# B&R Automation Studio project DivDiag
Automation Studio 4.9.2.46; technology packages: mapp 5.14.0, mappCockpit 5.14.0, mappMotion 5.14.0, mappView 5.14.0

## Configuration APC_XRAY

CPU PC_any, AutomationRuntime C4.72, Build 4.1.2, Safety 0.0, Vc V4.72.0

### Task classes (Cpu.sw)
```
Cyclic#1 (cycle 1600 us, tolerance 0 us):
  MainTest <- Source.MainTest.prg
  Maint <- Source.Diagnostic.Maint.prg
Cyclic#8 (cycle 9600 us):
  Vis <- Source.Vis.prg
DataObjects: McAcpSys
Binaries: mCoWebSc, FWRules, TCData, udbdef, mvLoader, McAcpSim, arsvcreg, McAcpDrv, arflatprv, arcoal, arconfig, Role, User, Cfg_Sec, asfw, iomap, Cfg_Sh, ashwd, ashwac, Cfg_PpList, sysconf, Cfg_Trak, McProfGen, TCLang, Cfg_Aut, Cfg_PVirt, Cfg_Ax, asnxdb1, Settings, CfgRec, Cfg_App2, Cfg_Comp, Cfg_Auto, Cfg_App1, Cfg_Set, TC, asnxdb2, AlarmCfg, AlarmHist, SSLCfg, Cfg_App6, Cfg_App5, Cfg_App4, Cfg_App3, AuditCfg, Cfg_Coupl, vccdt, vccline, vcfile, arial, vccbmp, vccstr, vcctrend, vcbclass, vcgclass, vcdsint, vcnet, vcshared, vcmgr, arialbd, vcxml, vccnum, vccbtn, vccovl, vccalarm, vccurl, vccslider, vccbar, vcctext, Visu01, Visu03, vcpdsw, vcfntttf, vcalarm, Visu02, vcrt, vcchtml, vcdsloc, vcchspot, vctcal, vcpdvnc, vcpfar00, vcpfmtcx, vcptelo, vcpdihd, vcpdi855, vcpfapc, vcpfppc7, vcpdi815, vcpk, Config_1, Config_4, Config_3, Config_2, CfgAlrm
Libraries: standard, AsBrStr, McAcpPar, McBase, sys_lib, runtime, arssl, fileio, mcacptrak, astime, asieccon, powerlnk, mcaxis, dataobj, aruser, mpaudit, vcresman, AsIODiag
```

### Hardware
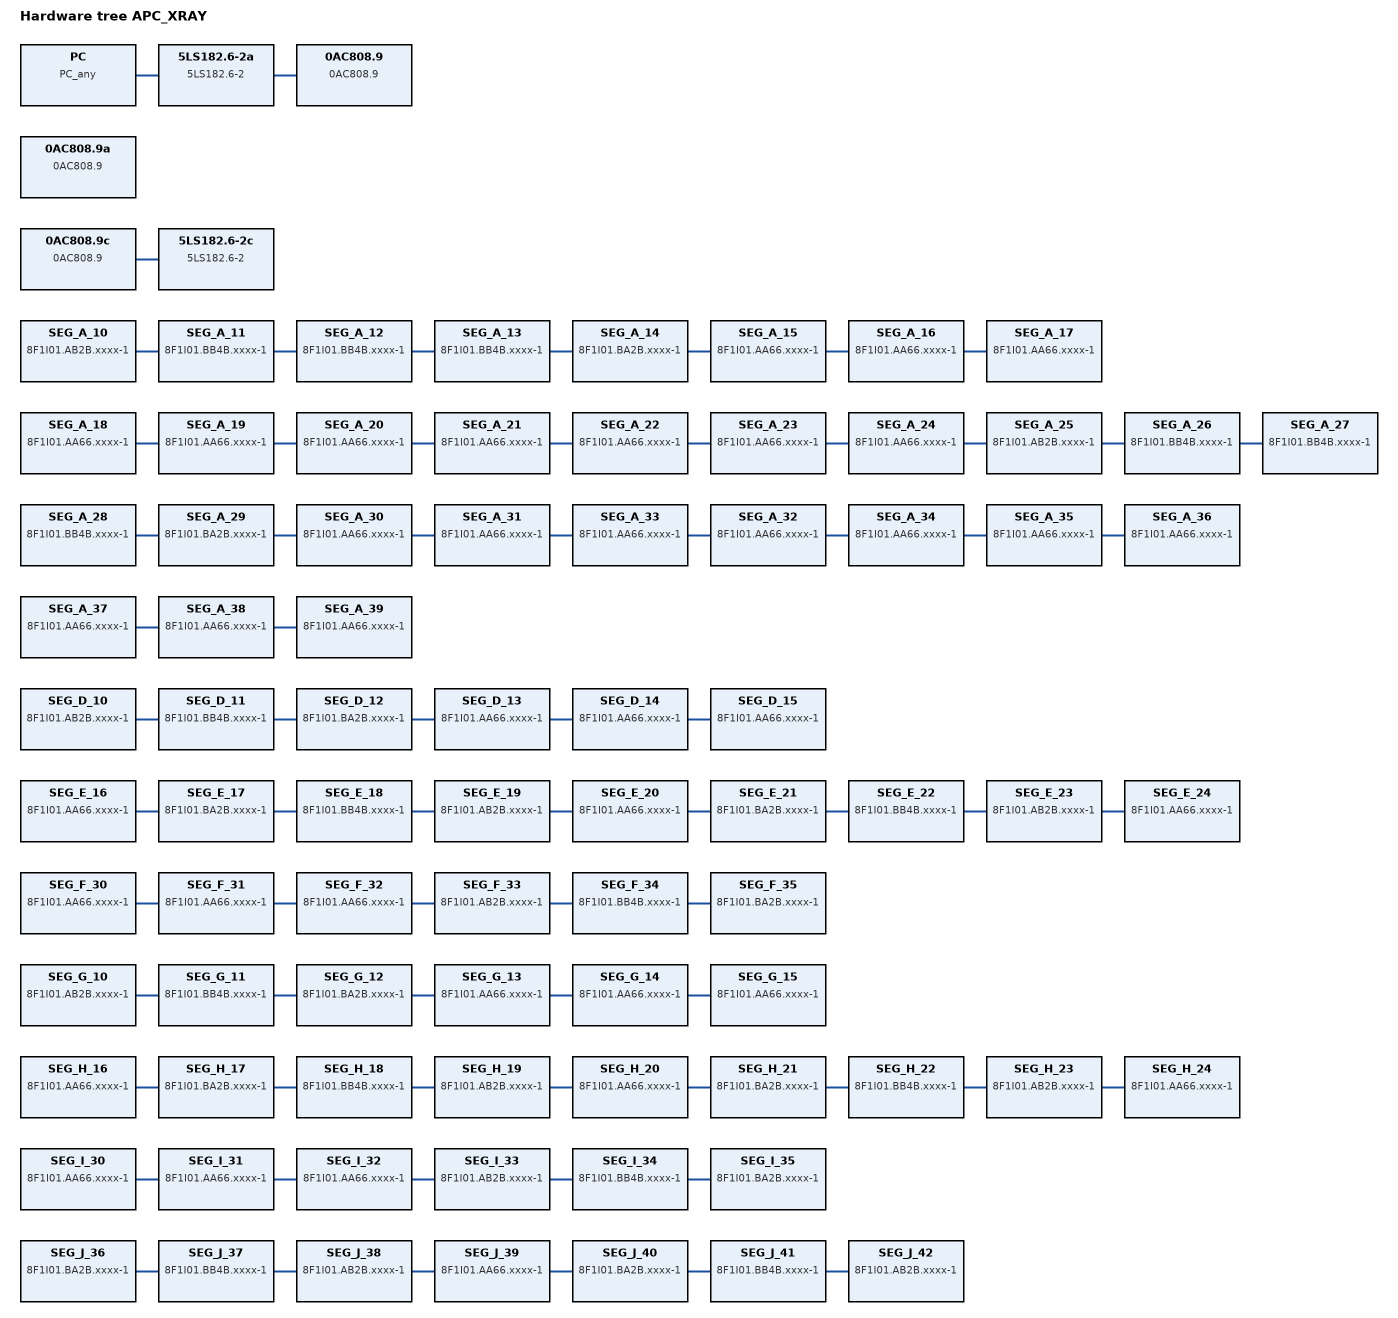
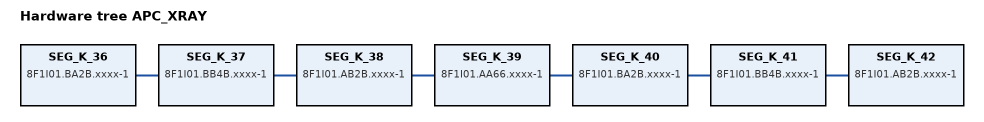
```
0AC808.9 : 0AC808.9 v1.0.0.0  [ETH1 -> 5LS182.6-2a.IF1 [Cable Type=PowerlinkCable, Length=10, Version=1.0.0.3]; ETH2 -> SEG_A_12.PLK3 [Cable Type=PowerlinkCable, Length=10, Version=1.0.0.3]; ETH3 -> SEG_A_22.PLK3 [Cable Type=PowerlinkCable, Length=10, Version=1.0.0.3]; ETH4 -> SEG_A_32.PLK3 [Cable Type=PowerlinkCable, Length=10, Version=1.0.0.3]]
0AC808.9a : 0AC808.9 v1.0.0.0  [ETH1 -> 5LS182.6-2c.IF1 [Cable Type=PowerlinkCable, Length=10, Version=1.0.0.3]; ETH2 -> SEG_G_10.PLK3 [Cable Type=PowerlinkCable, Length=10, Version=1.0.0.3]; ETH3 -> SEG_H_20.PLK3 [Cable Type=PowerlinkCable, Length=10, Version=1.0.0.3]; ETH4 -> SEG_I_35.PLK3 [Cable Type=PowerlinkCable, Length=10, Version=1.0.0.3]; ETH6 -> SEG_K_39.PLK3 [Cable Type=PowerlinkCable, Length=10, Version=1.0.0.3]]
0AC808.9c : 0AC808.9 v1.0.0.0  [ETH1 -> 5LS182.6-2c.PLK2 [Cable Type=PowerlinkCable, Length=10, Version=1.0.0.3]; ETH2 -> SEG_D_10.PLK3 [Cable Type=PowerlinkCable, Length=10, Version=1.0.0.3]; ETH3 -> SEG_E_20.PLK3 [Cable Type=PowerlinkCable, Length=10, Version=1.0.0.3]; ETH4 -> SEG_F_35.PLK3 [Cable Type=PowerlinkCable, Length=10, Version=1.0.0.3]; ETH6 -> SEG_J_39.PLK3 [Cable Type=PowerlinkCable, Length=10, Version=1.0.0.3]]
5LS182.6-2a : 5LS182.6-2 v1.7.1.0  [SL -> PC.SL1]
  Connector IF1:
    MtuSize = 1500
    DNAConfiguration = manual
    CycleTime = 1600
    EplNatSubnet = 192.168.102.0
  Supervision = off
5LS182.6-2c : 5LS182.6-2 v1.7.1.0  [PLK2 -> 0AC808.9c.ETH1 [Cable Type=PowerlinkCable, Length=10, Version=1.0.0.3]; SL -> PC.SL2]
  Connector IF1:
    DNAConfiguration = manual
    CycleTime = 1600
    NodeDefinition = Software
    EplNatSubnet = 192.168.104.0
PC : PC_any v1.1.1.0 (OrderNumber=PC)
  Connector IF1:
    ActivateDevice = 1
    ActivateIna = 1
    DeviceParam = /IR=4 /IO=0x3F8 /CLK=1843200 /IF=1
  Connector IF3:
    InaPort = 11159
  ConfigurationID = Starwheel_XRAY
  ConfigVersion = 1.0.2
  UserPartitionSize = 100
  UserRamSize = 250000
  RemMemSize = 250000
  PermanentPvSize = 10000
  RemanentGlobalPvSize = 10000
  VolatileGlobalPvSize = 100000
  SystemTick = 1600
  TaskClassIdleTime = 1600
  Cyclic1Duration = 1600
  Cyclic1Tolerance = 0
  Cyclic1Stack = 256000
  Cyclic2Duration = 19200
  Cyclic2Tolerance = 19200
  Cyclic3Duration = 49600
  Cyclic3Tolerance = 49600
  Cyclic4Duration = 99200
  Cyclic4Tolerance = 99200
  Cyclic6Duration = 499200
  Cyclic6Tolerance = 499200
  Cyclic8Duration = 9600
  FileDevice1
  FileDeviceName1 = SvgData
  FileDevicePath1 = ../../../../Logical/Scene/Generated
  FtpUser1
  FtpUsername1 = BnR
  FtpUserPassword1 = OwgnRUL028A/e+iGXLfM2NhZbf3ZfVOTPAeyn0eidZE=  // password
  FtpUserSalt1 = LWczKOmt
  FTPAccessRight1 = 0
  ActivateOpcUa = 1
  OpcUaInformationModels_PV_Version = 1
SEG_A_10 : 8F1I01.AB2B.xxxx-1 v1.0.0.2  [PLK1 -> SEG_A_39.PLK2 (NodeNumber=10) [Cable Type=PowerlinkCable, Length=10, Version=1.0.0.3]; PLK2 -> SEG_A_11.PLK1 (NodeNumber=10) [Cable Type=PowerlinkCable, Length=10, Version=1.0.0.3]]
  EnableDNA = on
  EPL_DNA_Head = 0
  EPL_DNA_Predecessor = 11
  EPL_DNA_HubPort = 1
  EPL_DNA_InPort = 2
  DriveConfiguration:
    McTypeID = LLMConfig
  DriveConfiguration/Segment:
    Shape = STRAIGHT105_TO_CIRCULAR
    SegmentReference = SEG_A_10
    StopReaction = UseAssemblySetting
    SpeedFilter = UseAssemblySetting
SEG_A_11 : 8F1I01.BB4B.xxxx-1 v1.0.0.2  [PLK1 -> SEG_A_10.PLK2 (NodeNumber=11) [Cable Type=PowerlinkCable, Length=10, Version=1.0.0.3]; PLK2 -> SEG_A_12.PLK1 (NodeNumber=11) [Cable Type=PowerlinkCable, Length=10, Version=1.0.0.3]]
  EnableDNA = on
  EPL_DNA_Head = 0
  EPL_DNA_Predecessor = 12
  EPL_DNA_HubPort = 1
  EPL_DNA_InPort = 2
  DriveConfiguration:
    McTypeID = LLMConfig
  DriveConfiguration/Segment:
    Shape = CIRCULAR
    SegmentReference = SEG_A_11
    StopReaction = UseAssemblySetting
    SpeedFilter = UseAssemblySetting
SEG_A_12 : 8F1I01.BB4B.xxxx-1 v1.0.0.2  [PLK1 -> SEG_A_11.PLK2 (NodeNumber=12) [Cable Type=PowerlinkCable, Length=10, Version=1.0.0.3]; PLK2 -> SEG_A_13.PLK1 (NodeNumber=12) [Cable Type=PowerlinkCable, Length=10, Version=1.0.0.3]; PLK3 -> 0AC808.9.ETH2 (NodeNumber=12) [Cable Type=PowerlinkCable, Length=10, Version=1.0.0.3]]
  EnableDNA = on
  EPL_DNA_Head = 0
  EPL_DNA_HubPort = 0
  EPL_DNA_InPort = 3
  DriveConfiguration:
    McTypeID = LLMConfig
  DriveConfiguration/Segment:
    Shape = CIRCULAR
    SegmentReference = SEG_A_12
    StopReaction = UseAssemblySetting
    SpeedFilter = UseAssemblySetting
SEG_A_13 : 8F1I01.BB4B.xxxx-1 v1.0.0.2  [PLK1 -> SEG_A_12.PLK2 (NodeNumber=13) [Cable Type=PowerlinkCable, Length=10, Version=1.0.0.3]; PLK2 -> SEG_A_14.PLK1 (NodeNumber=13) [Cable Type=PowerlinkCable, Length=10, Version=1.0.0.3]]
  EnableDNA = on
  EPL_DNA_Head = 0
  EPL_DNA_Predecessor = 12
  DriveConfiguration:
    McTypeID = LLMConfig
  DriveConfiguration/Segment:
    Shape = CIRCULAR
    SegmentReference = SEG_A_13
    StopReaction = UseAssemblySetting
    SpeedFilter = UseAssemblySetting
SEG_A_14 : 8F1I01.BA2B.xxxx-1 v1.0.0.2  [PLK1 -> SEG_A_13.PLK2 (NodeNumber=14) [Cable Type=PowerlinkCable, Length=10, Version=1.0.0.3]; PLK2 -> SEG_A_15.PLK1 (NodeNumber=14) [Cable Type=PowerlinkCable, Length=10, Version=1.0.0.3]]
  EnableDNA = on
  EPL_DNA_Head = 0
  EPL_DNA_Predecessor = 13
  DriveConfiguration:
    McTypeID = LLMConfig
  DriveConfiguration/Segment:
    Shape = CIRCULAR_TO_STRAIGHT105
    SegmentReference = SEG_A_14
    StopReaction = UseAssemblySetting
    SpeedFilter = UseAssemblySetting
SEG_A_15 : 8F1I01.AA66.xxxx-1 v1.0.0.2  [PLK1 -> SEG_A_14.PLK2 (NodeNumber=15) [Cable Type=PowerlinkCable, Length=10, Version=1.0.0.3]; PLK2 -> SEG_A_16.PLK1 (NodeNumber=15) [Cable Type=PowerlinkCable, Length=10, Version=1.0.0.3]]
  EnableDNA = on
  EPL_DNA_Head = 0
  EPL_DNA_Predecessor = 14
  DriveConfiguration:
    McTypeID = LLMConfig
  DriveConfiguration/Segment:
    Shape = STRAIGHT660
    SegmentReference = SEG_A_15
    StopReaction = UseAssemblySetting
    SpeedFilter = UseAssemblySetting
SEG_A_16 : 8F1I01.AA66.xxxx-1 v1.0.0.2  [PLK1 -> SEG_A_15.PLK2 (NodeNumber=16) [Cable Type=PowerlinkCable, Length=10, Version=1.0.0.3]; PLK2 -> SEG_A_17.PLK1 (NodeNumber=16) [Cable Type=PowerlinkCable, Length=10, Version=1.0.0.3]]
  EnableDNA = on
  EPL_DNA_Head = 0
  EPL_DNA_Predecessor = 15
  DriveConfiguration:
    McTypeID = LLMConfig
  DriveConfiguration/Segment:
    Shape = STRAIGHT660
    SegmentReference = SEG_A_16
    StopReaction = UseAssemblySetting
    SpeedFilter = UseAssemblySetting
SEG_A_17 : 8F1I01.AA66.xxxx-1 v1.0.0.2  [PLK1 -> SEG_A_16.PLK2 (NodeNumber=17) [Cable Type=PowerlinkCable, Length=10, Version=1.0.0.3]]
  EnableDNA = on
  EPL_DNA_Head = 0
  EPL_DNA_Predecessor = 16
  DriveConfiguration:
    McTypeID = LLMConfig
  DriveConfiguration/Segment:
    Shape = STRAIGHT660
    SegmentReference = SEG_A_17
    StopReaction = UseAssemblySetting
    SpeedFilter = UseAssemblySetting
SEG_A_18 : 8F1I01.AA66.xxxx-1 v1.0.0.2  [PLK2 -> SEG_A_19.PLK1 (NodeNumber=18) [Cable Type=PowerlinkCable, Length=10, Version=1.0.0.3]]
  EnableDNA = on
  EPL_DNA_Head = 0
  EPL_DNA_Predecessor = 19
  EPL_DNA_HubPort = 1
  EPL_DNA_InPort = 2
  DriveConfiguration:
    McTypeID = LLMConfig
  DriveConfiguration/Segment:
    Shape = STRAIGHT660
    SegmentReference = SEG_A_18
    StopReaction = UseAssemblySetting
    SpeedFilter = UseAssemblySetting
SEG_A_19 : 8F1I01.AA66.xxxx-1 v1.0.0.2  [PLK1 -> SEG_A_18.PLK2 (NodeNumber=19) [Cable Type=PowerlinkCable, Length=10, Version=1.0.0.3]; PLK2 -> SEG_A_20.PLK1 (NodeNumber=19) [Cable Type=PowerlinkCable, Length=10, Version=1.0.0.3]]
  EnableDNA = on
  EPL_DNA_Head = 0
  EPL_DNA_Predecessor = 20
  EPL_DNA_HubPort = 1
  EPL_DNA_InPort = 2
  DriveConfiguration:
    McTypeID = LLMConfig
  DriveConfiguration/Segment:
    Shape = STRAIGHT660
    SegmentReference = SEG_A_19
    StopReaction = UseAssemblySetting
    SpeedFilter = UseAssemblySetting
SEG_A_20 : 8F1I01.AA66.xxxx-1 v1.0.0.2  [PLK1 -> SEG_A_19.PLK2 (NodeNumber=20) [Cable Type=PowerlinkCable, Length=10, Version=1.0.0.3]; PLK2 -> SEG_A_21.PLK1 (NodeNumber=20) [Cable Type=PowerlinkCable, Length=10, Version=1.0.0.3]]
  EnableDNA = on
  EPL_DNA_Head = 0
  EPL_DNA_Predecessor = 21
  EPL_DNA_HubPort = 1
  EPL_DNA_InPort = 2
  DriveConfiguration:
    McTypeID = LLMConfig
  DriveConfiguration/Segment:
    Shape = STRAIGHT660
    SegmentReference = SEG_A_20
    StopReaction = UseAssemblySetting
    SpeedFilter = UseAssemblySetting
SEG_A_21 : 8F1I01.AA66.xxxx-1 v1.0.0.2  [PLK1 -> SEG_A_20.PLK2 (NodeNumber=21) [Cable Type=PowerlinkCable, Length=10, Version=1.0.0.3]; PLK2 -> SEG_A_22.PLK1 (NodeNumber=21) [Cable Type=PowerlinkCable, Length=10, Version=1.0.0.3]]
  EnableDNA = on
  EPL_DNA_Head = 0
  EPL_DNA_Predecessor = 22
  EPL_DNA_HubPort = 1
  EPL_DNA_InPort = 2
  DriveConfiguration:
    McTypeID = LLMConfig
  DriveConfiguration/Segment:
    Shape = STRAIGHT660
    SegmentReference = SEG_A_21
    StopReaction = UseAssemblySetting
    SpeedFilter = UseAssemblySetting
SEG_A_22 : 8F1I01.AA66.xxxx-1 v1.0.0.2  [PLK1 -> SEG_A_21.PLK2 (NodeNumber=22) [Cable Type=PowerlinkCable, Length=10, Version=1.0.0.3]; PLK2 -> SEG_A_23.PLK1 (NodeNumber=22) [Cable Type=PowerlinkCable, Length=10, Version=1.0.0.3]; PLK3 -> 0AC808.9.ETH3 (NodeNumber=22) [Cable Type=PowerlinkCable, Length=10, Version=1.0.0.3]]
  EnableDNA = on
  EPL_DNA_Head = 0
  EPL_DNA_HubPort = 0
  EPL_DNA_InPort = 3
  DriveConfiguration:
    McTypeID = LLMConfig
  DriveConfiguration/Segment:
    Shape = STRAIGHT660
    SegmentReference = SEG_A_22
    StopReaction = UseAssemblySetting
    SpeedFilter = UseAssemblySetting
SEG_A_23 : 8F1I01.AA66.xxxx-1 v1.0.0.2  [PLK1 -> SEG_A_22.PLK2 (NodeNumber=23) [Cable Type=PowerlinkCable, Length=10, Version=1.0.0.3]; PLK2 -> SEG_A_24.PLK1 (NodeNumber=23) [Cable Type=PowerlinkCable, Length=10, Version=1.0.0.3]]
  EnableDNA = on
  EPL_DNA_Head = 0
  EPL_DNA_Predecessor = 22
  DriveConfiguration:
    McTypeID = LLMConfig
  DriveConfiguration/Segment:
    Shape = STRAIGHT660
    SegmentReference = SEG_A_23
    StopReaction = UseAssemblySetting
    SpeedFilter = UseAssemblySetting
SEG_A_24 : 8F1I01.AA66.xxxx-1 v1.0.0.2  [PLK1 -> SEG_A_23.PLK2 (NodeNumber=24) [Cable Type=PowerlinkCable, Length=10, Version=1.0.0.3]; PLK2 -> SEG_A_25.PLK1 (NodeNumber=24) [Cable Type=PowerlinkCable, Length=10, Version=1.0.0.3]]
  EnableDNA = on
  EPL_DNA_Head = 0
  EPL_DNA_Predecessor = 23
  DriveConfiguration:
    McTypeID = LLMConfig
  DriveConfiguration/Segment:
    Shape = STRAIGHT660
    SegmentReference = SEG_A_24
    StopReaction = UseAssemblySetting
    SpeedFilter = UseAssemblySetting
SEG_A_25 : 8F1I01.AB2B.xxxx-1 v1.0.0.2  [PLK1 -> SEG_A_24.PLK2 (NodeNumber=25) [Cable Type=PowerlinkCable, Length=10, Version=1.0.0.3]; PLK2 -> SEG_A_26.PLK1 (NodeNumber=25) [Cable Type=PowerlinkCable, Length=10, Version=1.0.0.3]]
  EnableDNA = on
  EPL_DNA_Head = 0
  EPL_DNA_Predecessor = 24
  DriveConfiguration:
    McTypeID = LLMConfig
  DriveConfiguration/Segment:
    Shape = STRAIGHT105_TO_CIRCULAR
    SegmentReference = SEG_A_25
    StopReaction = UseAssemblySetting
    SpeedFilter = UseAssemblySetting
SEG_A_26 : 8F1I01.BB4B.xxxx-1 v1.0.0.2  [PLK1 -> SEG_A_25.PLK2 (NodeNumber=26) [Cable Type=PowerlinkCable, Length=10, Version=1.0.0.3]; PLK2 -> SEG_A_27.PLK1 (NodeNumber=26) [Cable Type=PowerlinkCable, Length=10, Version=1.0.0.3]]
  EnableDNA = on
  EPL_DNA_Head = 0
  EPL_DNA_Predecessor = 25
  DriveConfiguration:
    McTypeID = LLMConfig
  DriveConfiguration/Segment:
    Shape = CIRCULAR
    SegmentReference = SEG_A_26
    StopReaction = UseAssemblySetting
    SpeedFilter = UseAssemblySetting
SEG_A_27 : 8F1I01.BB4B.xxxx-1 v1.0.0.2  [PLK1 -> SEG_A_26.PLK2 (NodeNumber=27) [Cable Type=PowerlinkCable, Length=10, Version=1.0.0.3]]
  EnableDNA = on
  EPL_DNA_Head = 0
  EPL_DNA_Predecessor = 26
  DriveConfiguration:
    McTypeID = LLMConfig
  DriveConfiguration/Segment:
    Shape = CIRCULAR
    SegmentReference = SEG_A_27
    StopReaction = UseAssemblySetting
    SpeedFilter = UseAssemblySetting
SEG_A_28 : 8F1I01.BB4B.xxxx-1 v1.0.0.2  [PLK2 -> SEG_A_29.PLK1 (NodeNumber=28) [Cable Type=PowerlinkCable, Length=10, Version=1.0.0.3]]
  EnableDNA = on
  EPL_DNA_Head = 0
  EPL_DNA_Predecessor = 29
  EPL_DNA_HubPort = 1
  EPL_DNA_InPort = 2
  DriveConfiguration:
    McTypeID = LLMConfig
  DriveConfiguration/Segment:
    Shape = CIRCULAR
    SegmentReference = SEG_A_28
    StopReaction = UseAssemblySetting
    SpeedFilter = UseAssemblySetting
SEG_A_29 : 8F1I01.BA2B.xxxx-1 v1.0.0.2  [PLK1 -> SEG_A_28.PLK2 (NodeNumber=29) [Cable Type=PowerlinkCable, Length=10, Version=1.0.0.3]; PLK2 -> SEG_A_30.PLK1 (NodeNumber=29) [Cable Type=PowerlinkCable, Length=10, Version=1.0.0.3]]
  EnableDNA = on
  EPL_DNA_Head = 0
  EPL_DNA_Predecessor = 30
  EPL_DNA_HubPort = 1
  EPL_DNA_InPort = 2
  DriveConfiguration:
    McTypeID = LLMConfig
  DriveConfiguration/Segment:
    Shape = CIRCULAR_TO_STRAIGHT105
    SegmentReference = SEG_A_29
    StopReaction = UseAssemblySetting
    SpeedFilter = UseAssemblySetting
SEG_A_30 : 8F1I01.AA66.xxxx-1 v1.0.0.2  [PLK1 -> SEG_A_29.PLK2 (NodeNumber=30) [Cable Type=PowerlinkCable, Length=10, Version=1.0.0.3]; PLK2 -> SEG_A_31.PLK1 (NodeNumber=30) [Cable Type=PowerlinkCable, Length=10, Version=1.0.0.3]]
  EnableDNA = on
  EPL_DNA_Head = 0
  EPL_DNA_Predecessor = 31
  EPL_DNA_HubPort = 1
  EPL_DNA_InPort = 2
  DriveConfiguration:
    McTypeID = LLMConfig
  DriveConfiguration/Segment:
    Shape = STRAIGHT660
    SegmentReference = SEG_A_30
    StopReaction = UseAssemblySetting
    SpeedFilter = UseAssemblySetting
SEG_A_31 : 8F1I01.AA66.xxxx-1 v1.0.0.2  [PLK1 -> SEG_A_30.PLK2 (NodeNumber=31) [Cable Type=PowerlinkCable, Length=10, Version=1.0.0.3]; PLK2 -> SEG_A_33.PLK1 (NodeNumber=31) [Cable Type=PowerlinkCable, Length=10, Version=1.0.0.3]]
  EnableDNA = on
  EPL_DNA_Head = 0
  EPL_DNA_Predecessor = 32
  EPL_DNA_HubPort = 1
  EPL_DNA_InPort = 2
  DriveConfiguration:
    McTypeID = LLMConfig
  DriveConfiguration/Segment:
    Shape = STRAIGHT660
    SegmentReference = SEG_A_31
    StopReaction = UseAssemblySetting
    SpeedFilter = UseAssemblySetting
SEG_A_32 : 8F1I01.AA66.xxxx-1 v1.0.0.2  [PLK1 -> SEG_A_33.PLK2 (NodeNumber=32) [Cable Type=PowerlinkCable, Length=10, Version=1.0.0.3]; PLK2 -> SEG_A_34.PLK1 (NodeNumber=32) [Cable Type=PowerlinkCable, Length=10, Version=1.0.0.3]; PLK3 -> 0AC808.9.ETH4 (NodeNumber=32) [Cable Type=PowerlinkCable, Length=10, Version=1.0.0.3]]
  EnableDNA = on
  EPL_DNA_Head = 0
  EPL_DNA_HubPort = 0
  EPL_DNA_InPort = 3
  DriveConfiguration:
    McTypeID = LLMConfig
  DriveConfiguration/Segment:
    Shape = STRAIGHT660
    SegmentReference = SEG_A_32
    StopReaction = UseAssemblySetting
    SpeedFilter = UseAssemblySetting
SEG_A_33 : 8F1I01.AA66.xxxx-1 v1.0.0.2  [PLK1 -> SEG_A_31.PLK2 (NodeNumber=33) [Cable Type=PowerlinkCable, Length=10, Version=1.0.0.3]; PLK2 -> SEG_A_32.PLK1 (NodeNumber=33) [Cable Type=PowerlinkCable, Length=10, Version=1.0.0.3]]
  EnableDNA = on
  EPL_DNA_Head = 0
  EPL_DNA_Predecessor = 32
  DriveConfiguration:
    McTypeID = LLMConfig
  DriveConfiguration/Segment:
    Shape = STRAIGHT660
    SegmentReference = SEG_A_33
    StopReaction = UseAssemblySetting
    SpeedFilter = UseAssemblySetting
SEG_A_34 : 8F1I01.AA66.xxxx-1 v1.0.0.2  [PLK1 -> SEG_A_32.PLK2 (NodeNumber=34) [Cable Type=PowerlinkCable, Length=10, Version=1.0.0.3]; PLK2 -> SEG_A_35.PLK1 (NodeNumber=34) [Cable Type=PowerlinkCable, Length=10, Version=1.0.0.3]]
  EnableDNA = on
  EPL_DNA_Head = 0
  EPL_DNA_Predecessor = 33
  DriveConfiguration:
    McTypeID = LLMConfig
  DriveConfiguration/Segment:
    Shape = STRAIGHT660
    SegmentReference = SEG_A_34
    StopReaction = UseAssemblySetting
    SpeedFilter = UseAssemblySetting
SEG_A_35 : 8F1I01.AA66.xxxx-1 v1.0.0.2  [PLK1 -> SEG_A_34.PLK2 (NodeNumber=35) [Cable Type=PowerlinkCable, Length=10, Version=1.0.0.3]; PLK2 -> SEG_A_36.PLK1 (NodeNumber=35) [Cable Type=PowerlinkCable, Length=10, Version=1.0.0.3]]
  EnableDNA = on
  EPL_DNA_Head = 0
  EPL_DNA_Predecessor = 34
  DriveConfiguration:
    McTypeID = LLMConfig
  DriveConfiguration/Segment:
    Shape = STRAIGHT660
    SegmentReference = SEG_A_35
    StopReaction = UseAssemblySetting
    SpeedFilter = UseAssemblySetting
SEG_A_36 : 8F1I01.AA66.xxxx-1 v1.0.0.2  [PLK1 -> SEG_A_35.PLK2 (NodeNumber=36) [Cable Type=PowerlinkCable, Length=10, Version=1.0.0.3]]
  EnableDNA = on
  EPL_DNA_Head = 0
  EPL_DNA_Predecessor = 35
  DriveConfiguration:
    McTypeID = LLMConfig
  DriveConfiguration/Segment:
    Shape = STRAIGHT660
    SegmentReference = SEG_A_36
    StopReaction = UseAssemblySetting
    SpeedFilter = UseAssemblySetting
SEG_A_37 : 8F1I01.AA66.xxxx-1 v1.0.0.2  [PLK2 -> SEG_A_38.PLK1 (NodeNumber=37) [Cable Type=PowerlinkCable, Length=10, Version=1.0.0.3]]
  EnableDNA = on
  EPL_DNA_Head = 0
  EPL_DNA_Predecessor = 38
  EPL_DNA_HubPort = 1
  EPL_DNA_InPort = 2
  DriveConfiguration:
    McTypeID = LLMConfig
  DriveConfiguration/Segment:
    Shape = STRAIGHT660
    SegmentReference = SEG_A_37
    StopReaction = UseAssemblySetting
    SpeedFilter = UseAssemblySetting
SEG_A_38 : 8F1I01.AA66.xxxx-1 v1.0.0.2  [PLK1 -> SEG_A_37.PLK2 (NodeNumber=38) [Cable Type=PowerlinkCable, Length=10, Version=1.0.0.3]; PLK2 -> SEG_A_39.PLK1 (NodeNumber=38) [Cable Type=PowerlinkCable, Length=10, Version=1.0.0.3]]
  EnableDNA = on
  EPL_DNA_Head = 0
  EPL_DNA_Predecessor = 39
  EPL_DNA_HubPort = 1
  EPL_DNA_InPort = 2
  DriveConfiguration:
    McTypeID = LLMConfig
  DriveConfiguration/Segment:
    Shape = STRAIGHT660
    SegmentReference = SEG_A_38
    StopReaction = UseAssemblySetting
    SpeedFilter = UseAssemblySetting
SEG_A_39 : 8F1I01.AA66.xxxx-1 v1.0.0.2  [PLK1 -> SEG_A_38.PLK2 (NodeNumber=39) [Cable Type=PowerlinkCable, Length=10, Version=1.0.0.3]; PLK2 -> SEG_A_10.PLK1 (NodeNumber=39) [Cable Type=PowerlinkCable, Length=10, Version=1.0.0.3]]
  EnableDNA = on
  EPL_DNA_Head = 0
  EPL_DNA_Predecessor = 10
  EPL_DNA_HubPort = 1
  EPL_DNA_InPort = 2
  DriveConfiguration:
    McTypeID = LLMConfig
  DriveConfiguration/Segment:
    Shape = STRAIGHT660
    SegmentReference = SEG_A_39
    StopReaction = UseAssemblySetting
    SpeedFilter = UseAssemblySetting
SEG_D_10 : 8F1I01.AB2B.xxxx-1 v1.0.0.2  [PLK2 -> SEG_D_11.PLK1 (NodeNumber=3) [Cable Type=PowerlinkCable, Length=10, Version=1.0.0.3]; PLK3 -> 0AC808.9c.ETH2 (NodeNumber=3) [Cable Type=PowerlinkCable, Length=10, Version=1.0.0.3]]
  EnableDNA = on
  EPL_DNA_Head = 0
  EPL_DNA_HubPort = 0
  EPL_DNA_InPort = 3
  DriveConfiguration:
    McTypeID = LLMConfig
  DriveConfiguration/Segment:
    Shape = STRAIGHT105_TO_CIRCULAR
    SegmentReference = SEG_D_10
    StopReaction = UseAssemblySetting
    SpeedFilter = UseAssemblySetting
SEG_D_11 : 8F1I01.BB4B.xxxx-1 v1.0.0.2  [PLK1 -> SEG_D_10.PLK2 (NodeNumber=4) [Cable Type=PowerlinkCable, Length=10, Version=1.0.0.3]; PLK2 -> SEG_D_12.PLK1 (NodeNumber=4) [Cable Type=PowerlinkCable, Length=10, Version=1.0.0.3]]
  EnableDNA = on
  EPL_DNA_Head = 0
  EPL_DNA_Predecessor = 10
  DriveConfiguration:
    McTypeID = LLMConfig
  DriveConfiguration/Segment:
    Shape = CIRCULAR
    SegmentReference = SEG_D_11
    StopReaction = UseAssemblySetting
    SpeedFilter = UseAssemblySetting
SEG_D_12 : 8F1I01.BA2B.xxxx-1 v1.0.0.2  [PLK1 -> SEG_D_11.PLK2 (NodeNumber=5) [Cable Type=PowerlinkCable, Length=10, Version=1.0.0.3]; PLK2 -> SEG_D_13.PLK1 (NodeNumber=5) [Cable Type=PowerlinkCable, Length=10, Version=1.0.0.3]]
  EnableDNA = on
  EPL_DNA_Head = 0
  EPL_DNA_Predecessor = 11
  DriveConfiguration:
    McTypeID = LLMConfig
  DriveConfiguration/Segment:
    Shape = CIRCULAR_TO_STRAIGHT105
    SegmentReference = SEG_D_12
    StopReaction = UseAssemblySetting
    SpeedFilter = UseAssemblySetting
SEG_D_13 : 8F1I01.AA66.xxxx-1 v1.0.0.2  [PLK1 -> SEG_D_12.PLK2 (NodeNumber=6) [Cable Type=PowerlinkCable, Length=10, Version=1.0.0.3]; PLK2 -> SEG_D_14.PLK1 (NodeNumber=6) [Cable Type=PowerlinkCable, Length=10, Version=1.0.0.3]]
  EnableDNA = on
  EPL_DNA_Head = 0
  EPL_DNA_Predecessor = 12
  DriveConfiguration:
    McTypeID = LLMConfig
  DriveConfiguration/Segment:
    Shape = STRAIGHT660
    SegmentReference = SEG_D_13
    StopReaction = UseAssemblySetting
    SpeedFilter = UseAssemblySetting
SEG_D_14 : 8F1I01.AA66.xxxx-1 v1.0.0.2  [PLK1 -> SEG_D_13.PLK2 (NodeNumber=7) [Cable Type=PowerlinkCable, Length=10, Version=1.0.0.3]; PLK2 -> SEG_D_15.PLK1 (NodeNumber=7) [Cable Type=PowerlinkCable, Length=10, Version=1.0.0.3]]
  EnableDNA = on
  EPL_DNA_Head = 0
  EPL_DNA_Predecessor = 13
  DriveConfiguration:
    McTypeID = LLMConfig
  DriveConfiguration/Segment:
    Shape = STRAIGHT660
    SegmentReference = SEG_D_14
    StopReaction = UseAssemblySetting
    SpeedFilter = UseAssemblySetting
SEG_D_15 : 8F1I01.AA66.xxxx-1 v1.0.0.2  [PLK1 -> SEG_D_14.PLK2 (NodeNumber=8) [Cable Type=PowerlinkCable, Length=10, Version=1.0.0.3]]
  EnableDNA = on
  EPL_DNA_Head = 0
  EPL_DNA_Predecessor = 14
  DriveConfiguration:
    McTypeID = LLMConfig
  DriveConfiguration/Segment:
    Shape = STRAIGHT660
    SegmentReference = SEG_D_15
    StopReaction = UseAssemblySetting
    SpeedFilter = UseAssemblySetting
SEG_E_16 : 8F1I01.AA66.xxxx-1 v1.0.0.2  [PLK2 -> SEG_E_17.PLK1 (NodeNumber=28) [Cable Type=PowerlinkCable, Length=10, Version=1.0.0.3]]
  EnableDNA = on
  EPL_DNA_Head = 0
  EPL_DNA_Predecessor = 17
  DriveConfiguration:
    McTypeID = LLMConfig
  DriveConfiguration/Segment:
    Shape = STRAIGHT660
    SegmentReference = SEG_E_16
    StopReaction = UseAssemblySetting
    SpeedFilter = UseAssemblySetting
SEG_E_17 : 8F1I01.BA2B.xxxx-1 v1.0.0.2  [PLK1 -> SEG_E_16.PLK2 (NodeNumber=27) [Cable Type=PowerlinkCable, Length=10, Version=1.0.0.3]; PLK2 -> SEG_E_18.PLK1 (NodeNumber=27) [Cable Type=PowerlinkCable, Length=10, Version=1.0.0.3]]
  EnableDNA = on
  EPL_DNA_Head = 0
  EPL_DNA_Predecessor = 18
  DriveConfiguration:
    McTypeID = LLMConfig
  DriveConfiguration/Segment:
    Shape = CIRCULAR_TO_STRAIGHT105
    SegmentReference = SEG_E_17
    StopReaction = UseAssemblySetting
    SpeedFilter = UseAssemblySetting
SEG_E_18 : 8F1I01.BB4B.xxxx-1 v1.0.0.2  [PLK1 -> SEG_E_17.PLK2 (NodeNumber=26) [Cable Type=PowerlinkCable, Length=10, Version=1.0.0.3]; PLK2 -> SEG_E_19.PLK1 (NodeNumber=26) [Cable Type=PowerlinkCable, Length=10, Version=1.0.0.3]]
  EnableDNA = on
  EPL_DNA_Head = 0
  EPL_DNA_Predecessor = 19
  DriveConfiguration:
    McTypeID = LLMConfig
  DriveConfiguration/Segment:
    Shape = CIRCULAR
    SegmentReference = SEG_E_18
    StopReaction = UseAssemblySetting
    SpeedFilter = UseAssemblySetting
SEG_E_19 : 8F1I01.AB2B.xxxx-1 v1.0.0.2  [PLK1 -> SEG_E_18.PLK2 (NodeNumber=25) [Cable Type=PowerlinkCable, Length=10, Version=1.0.0.3]; PLK2 -> SEG_E_20.PLK1 (NodeNumber=25) [Cable Type=PowerlinkCable, Length=10, Version=1.0.0.3]]
  EnableDNA = on
  EPL_DNA_Head = 0
  EPL_DNA_Predecessor = 20
  DriveConfiguration:
    McTypeID = LLMConfig
  DriveConfiguration/Segment:
    Shape = STRAIGHT105_TO_CIRCULAR
    SegmentReference = SEG_E_19
    StopReaction = UseAssemblySetting
    SpeedFilter = UseAssemblySetting
SEG_E_20 : 8F1I01.AA66.xxxx-1 v1.0.0.2  [PLK1 -> SEG_E_19.PLK2 (NodeNumber=9) [Cable Type=PowerlinkCable, Length=10, Version=1.0.0.3]; PLK2 -> SEG_E_21.PLK1 (NodeNumber=9) [Cable Type=PowerlinkCable, Length=10, Version=1.0.0.3]; PLK3 -> 0AC808.9c.ETH3 (NodeNumber=9) [Cable Type=PowerlinkCable, Length=10, Version=1.0.0.3]]
  EnableDNA = on
  EPL_DNA_Head = 0
  EPL_DNA_HubPort = 0
  EPL_DNA_InPort = 3
  DriveConfiguration:
    McTypeID = LLMConfig
  DriveConfiguration/Segment:
    Shape = STRAIGHT660
    SegmentReference = SEG_E_20
    StopReaction = UseAssemblySetting
    SpeedFilter = UseAssemblySetting
SEG_E_21 : 8F1I01.BA2B.xxxx-1 v1.0.0.2  [PLK1 -> SEG_E_20.PLK2 (NodeNumber=29) [Cable Type=PowerlinkCable, Length=10, Version=1.0.0.3]; PLK2 -> SEG_E_22.PLK1 (NodeNumber=29) [Cable Type=PowerlinkCable, Length=10, Version=1.0.0.3]]
  EnableDNA = on
  EPL_DNA_Head = 0
  EPL_DNA_Predecessor = 20
  EPL_DNA_HubPort = 1
  EPL_DNA_InPort = 2
  DriveConfiguration:
    McTypeID = LLMConfig
  DriveConfiguration/Segment:
    Shape = CIRCULAR_TO_STRAIGHT105
    SegmentReference = SEG_E_21
    StopReaction = UseAssemblySetting
    SpeedFilter = UseAssemblySetting
SEG_E_22 : 8F1I01.BB4B.xxxx-1 v1.0.0.2  [PLK1 -> SEG_E_21.PLK2 (NodeNumber=43) [Cable Type=PowerlinkCable, Length=10, Version=1.0.0.3]; PLK2 -> SEG_E_23.PLK1 (NodeNumber=43) [Cable Type=PowerlinkCable, Length=10, Version=1.0.0.3]]
  EnableDNA = on
  EPL_DNA_Head = 0
  EPL_DNA_Predecessor = 21
  EPL_DNA_HubPort = 1
  EPL_DNA_InPort = 2
  DriveConfiguration:
    McTypeID = LLMConfig
  DriveConfiguration/Segment:
    Shape = CIRCULAR
    SegmentReference = SEG_E_22
    StopReaction = UseAssemblySetting
    SpeedFilter = UseAssemblySetting
SEG_E_23 : 8F1I01.AB2B.xxxx-1 v1.0.0.2  [PLK1 -> SEG_E_22.PLK2 (NodeNumber=44) [Cable Type=PowerlinkCable, Length=10, Version=1.0.0.3]; PLK2 -> SEG_E_24.PLK1 (NodeNumber=44) [Cable Type=PowerlinkCable, Length=10, Version=1.0.0.3]]
  EnableDNA = on
  EPL_DNA_Head = 0
  EPL_DNA_Predecessor = 22
  EPL_DNA_HubPort = 1
  EPL_DNA_InPort = 2
  DriveConfiguration:
    McTypeID = LLMConfig
  DriveConfiguration/Segment:
    Shape = STRAIGHT105_TO_CIRCULAR
    SegmentReference = SEG_E_23
    StopReaction = UseAssemblySetting
    SpeedFilter = UseAssemblySetting
SEG_E_24 : 8F1I01.AA66.xxxx-1 v1.0.0.2  [PLK1 -> SEG_E_23.PLK2 (NodeNumber=45) [Cable Type=PowerlinkCable, Length=10, Version=1.0.0.3]]
  EnableDNA = on
  EPL_DNA_Head = 0
  EPL_DNA_Predecessor = 23
  EPL_DNA_HubPort = 1
  EPL_DNA_InPort = 2
  DriveConfiguration:
    McTypeID = LLMConfig
  DriveConfiguration/Segment:
    Shape = STRAIGHT660
    SegmentReference = SEG_E_24
    StopReaction = UseAssemblySetting
    SpeedFilter = UseAssemblySetting
SEG_F_30 : 8F1I01.AA66.xxxx-1 v1.0.0.2  [PLK2 -> SEG_F_31.PLK1 (NodeNumber=51) [Cable Type=PowerlinkCable, Length=10, Version=1.0.0.3]]
  EnableDNA = on
  EPL_DNA_Head = 0
  EPL_DNA_Predecessor = 31
  EPL_DNA_HubPort = 1
  EPL_DNA_InPort = 2
  DriveConfiguration:
    McTypeID = LLMConfig
  DriveConfiguration/Segment:
    Shape = STRAIGHT660
    SegmentReference = SEG_F_30
    StopReaction = UseAssemblySetting
    SpeedFilter = UseAssemblySetting
SEG_F_31 : 8F1I01.AA66.xxxx-1 v1.0.0.2  [PLK1 -> SEG_F_30.PLK2 (NodeNumber=50) [Cable Type=PowerlinkCable, Length=10, Version=1.0.0.3]; PLK2 -> SEG_F_32.PLK1 (NodeNumber=50) [Cable Type=PowerlinkCable, Length=10, Version=1.0.0.3]]
  EnableDNA = on
  EPL_DNA_Head = 0
  EPL_DNA_Predecessor = 32
  EPL_DNA_HubPort = 1
  EPL_DNA_InPort = 2
  DriveConfiguration:
    McTypeID = LLMConfig
  DriveConfiguration/Segment:
    Shape = STRAIGHT660
    SegmentReference = SEG_F_31
    StopReaction = UseAssemblySetting
    SpeedFilter = UseAssemblySetting
SEG_F_32 : 8F1I01.AA66.xxxx-1 v1.0.0.2  [PLK1 -> SEG_F_31.PLK2 (NodeNumber=49) [Cable Type=PowerlinkCable, Length=10, Version=1.0.0.3]; PLK2 -> SEG_F_33.PLK1 (NodeNumber=49) [Cable Type=PowerlinkCable, Length=10, Version=1.0.0.3]]
  EnableDNA = on
  EPL_DNA_Head = 0
  EPL_DNA_Predecessor = 33
  EPL_DNA_HubPort = 1
  EPL_DNA_InPort = 2
  DriveConfiguration:
    McTypeID = LLMConfig
  DriveConfiguration/Segment:
    Shape = STRAIGHT660
    SegmentReference = SEG_F_32
    StopReaction = UseAssemblySetting
    SpeedFilter = UseAssemblySetting
SEG_F_33 : 8F1I01.AB2B.xxxx-1 v1.0.0.2  [PLK1 -> SEG_F_32.PLK2 (NodeNumber=48) [Cable Type=PowerlinkCable, Length=10, Version=1.0.0.3]; PLK2 -> SEG_F_34.PLK1 (NodeNumber=48) [Cable Type=PowerlinkCable, Length=10, Version=1.0.0.3]]
  EnableDNA = on
  EPL_DNA_Head = 0
  EPL_DNA_Predecessor = 34
  EPL_DNA_HubPort = 1
  EPL_DNA_InPort = 2
  DriveConfiguration:
    McTypeID = LLMConfig
  DriveConfiguration/Segment:
    Shape = STRAIGHT105_TO_CIRCULAR
    SegmentReference = SEG_F_33
    StopReaction = UseAssemblySetting
    SpeedFilter = UseAssemblySetting
SEG_F_34 : 8F1I01.BB4B.xxxx-1 v1.0.0.2  [PLK1 -> SEG_F_33.PLK2 (NodeNumber=47) [Cable Type=PowerlinkCable, Length=10, Version=1.0.0.3]; PLK2 -> SEG_F_35.PLK1 (NodeNumber=47) [Cable Type=PowerlinkCable, Length=10, Version=1.0.0.3]]
  EnableDNA = on
  EPL_DNA_Head = 0
  EPL_DNA_Predecessor = 35
  EPL_DNA_HubPort = 1
  EPL_DNA_InPort = 2
  DriveConfiguration:
    McTypeID = LLMConfig
  DriveConfiguration/Segment:
    Shape = CIRCULAR
    SegmentReference = SEG_F_34
    StopReaction = UseAssemblySetting
    SpeedFilter = UseAssemblySetting
SEG_F_35 : 8F1I01.BA2B.xxxx-1 v1.0.0.2  [PLK1 -> SEG_F_34.PLK2 (NodeNumber=46) [Cable Type=PowerlinkCable, Length=10, Version=1.0.0.3]; PLK3 -> 0AC808.9c.ETH4 (NodeNumber=46) [Cable Type=PowerlinkCable, Length=10, Version=1.0.0.3]]
  EnableDNA = on
  EPL_DNA_Head = 0
  EPL_DNA_HubPort = 0
  EPL_DNA_InPort = 3
  DriveConfiguration:
    McTypeID = LLMConfig
  DriveConfiguration/Segment:
    Shape = CIRCULAR_TO_STRAIGHT105
    SegmentReference = SEG_F_35
    StopReaction = UseAssemblySetting
    SpeedFilter = UseAssemblySetting
SEG_G_10 : 8F1I01.AB2B.xxxx-1 v1.0.0.2  [PLK2 -> SEG_G_11.PLK1 (NodeNumber=10) [Cable Type=PowerlinkCable, Length=10, Version=1.0.0.3]; PLK3 -> 0AC808.9a.ETH2 (NodeNumber=10) [Cable Type=PowerlinkCable, Length=10, Version=1.0.0.3]]
  EnableDNA = on
  EPL_DNA_Head = 0
  EPL_DNA_HubPort = 0
  EPL_DNA_InPort = 3
  DriveConfiguration:
    McTypeID = LLMConfig
  DriveConfiguration/Segment:
    Shape = STRAIGHT105_TO_CIRCULAR
    SegmentReference = SEG_G_10
    StopReaction = UseAssemblySetting
    SpeedFilter = UseAssemblySetting
SEG_G_11 : 8F1I01.BB4B.xxxx-1 v1.0.0.2  [PLK1 -> SEG_G_10.PLK2 (NodeNumber=11) [Cable Type=PowerlinkCable, Length=10, Version=1.0.0.3]; PLK2 -> SEG_G_12.PLK1 (NodeNumber=11) [Cable Type=PowerlinkCable, Length=10, Version=1.0.0.3]]
  EnableDNA = on
  EPL_DNA_Head = 0
  EPL_DNA_Predecessor = 10
  DriveConfiguration:
    McTypeID = LLMConfig
  DriveConfiguration/Segment:
    Shape = CIRCULAR
    SegmentReference = SEG_G_11
    StopReaction = UseAssemblySetting
    SpeedFilter = UseAssemblySetting
SEG_G_12 : 8F1I01.BA2B.xxxx-1 v1.0.0.2  [PLK1 -> SEG_G_11.PLK2 (NodeNumber=12) [Cable Type=PowerlinkCable, Length=10, Version=1.0.0.3]; PLK2 -> SEG_G_13.PLK1 (NodeNumber=12) [Cable Type=PowerlinkCable, Length=10, Version=1.0.0.3]]
  EnableDNA = on
  EPL_DNA_Head = 0
  EPL_DNA_Predecessor = 11
  DriveConfiguration:
    McTypeID = LLMConfig
  DriveConfiguration/Segment:
    Shape = CIRCULAR_TO_STRAIGHT105
    SegmentReference = SEG_G_12
    StopReaction = UseAssemblySetting
    SpeedFilter = UseAssemblySetting
SEG_G_13 : 8F1I01.AA66.xxxx-1 v1.0.0.2  [PLK1 -> SEG_G_12.PLK2 (NodeNumber=13) [Cable Type=PowerlinkCable, Length=10, Version=1.0.0.3]; PLK2 -> SEG_G_14.PLK1 (NodeNumber=13) [Cable Type=PowerlinkCable, Length=10, Version=1.0.0.3]]
  EnableDNA = on
  EPL_DNA_Head = 0
  EPL_DNA_Predecessor = 12
  DriveConfiguration:
    McTypeID = LLMConfig
  DriveConfiguration/Segment:
    Shape = STRAIGHT660
    SegmentReference = SEG_G_13
    StopReaction = UseAssemblySetting
    SpeedFilter = UseAssemblySetting
SEG_G_14 : 8F1I01.AA66.xxxx-1 v1.0.0.2  [PLK1 -> SEG_G_13.PLK2 (NodeNumber=14) [Cable Type=PowerlinkCable, Length=10, Version=1.0.0.3]; PLK2 -> SEG_G_15.PLK1 (NodeNumber=14) [Cable Type=PowerlinkCable, Length=10, Version=1.0.0.3]]
  EnableDNA = on
  EPL_DNA_Head = 0
  EPL_DNA_Predecessor = 13
  DriveConfiguration:
    McTypeID = LLMConfig
  DriveConfiguration/Segment:
    Shape = STRAIGHT660
    SegmentReference = SEG_G_14
    StopReaction = UseAssemblySetting
    SpeedFilter = UseAssemblySetting
SEG_G_15 : 8F1I01.AA66.xxxx-1 v1.0.0.2  [PLK1 -> SEG_G_14.PLK2 (NodeNumber=15) [Cable Type=PowerlinkCable, Length=10, Version=1.0.0.3]]
  EnableDNA = on
  EPL_DNA_Head = 0
  EPL_DNA_Predecessor = 14
  DriveConfiguration:
    McTypeID = LLMConfig
  DriveConfiguration/Segment:
    Shape = STRAIGHT660
    SegmentReference = SEG_G_15
    StopReaction = UseAssemblySetting
    SpeedFilter = UseAssemblySetting
SEG_H_16 : 8F1I01.AA66.xxxx-1 v1.0.0.2  [PLK2 -> SEG_H_17.PLK1 (NodeNumber=16) [Cable Type=PowerlinkCable, Length=10, Version=1.0.0.3]]
  EnableDNA = on
  EPL_DNA_Head = 0
  EPL_DNA_Predecessor = 17
  DriveConfiguration:
    McTypeID = LLMConfig
  DriveConfiguration/Segment:
    Shape = STRAIGHT660
    SegmentReference = SEG_H_16
    StopReaction = UseAssemblySetting
    SpeedFilter = UseAssemblySetting
SEG_H_17 : 8F1I01.BA2B.xxxx-1 v1.0.0.2  [PLK1 -> SEG_H_16.PLK2 (NodeNumber=17) [Cable Type=PowerlinkCable, Length=10, Version=1.0.0.3]; PLK2 -> SEG_H_18.PLK1 (NodeNumber=17) [Cable Type=PowerlinkCable, Length=10, Version=1.0.0.3]]
  EnableDNA = on
  EPL_DNA_Head = 0
  EPL_DNA_Predecessor = 18
  DriveConfiguration:
    McTypeID = LLMConfig
  DriveConfiguration/Segment:
    Shape = CIRCULAR_TO_STRAIGHT105
    SegmentReference = SEG_H_17
    StopReaction = UseAssemblySetting
    SpeedFilter = UseAssemblySetting
SEG_H_18 : 8F1I01.BB4B.xxxx-1 v1.0.0.2  [PLK1 -> SEG_H_17.PLK2 (NodeNumber=18) [Cable Type=PowerlinkCable, Length=10, Version=1.0.0.3]; PLK2 -> SEG_H_19.PLK1 (NodeNumber=18) [Cable Type=PowerlinkCable, Length=10, Version=1.0.0.3]]
  EnableDNA = on
  EPL_DNA_Head = 0
  EPL_DNA_Predecessor = 19
  DriveConfiguration:
    McTypeID = LLMConfig
  DriveConfiguration/Segment:
    Shape = CIRCULAR
    SegmentReference = SEG_H_18
    StopReaction = UseAssemblySetting
    SpeedFilter = UseAssemblySetting
SEG_H_19 : 8F1I01.AB2B.xxxx-1 v1.0.0.2  [PLK1 -> SEG_H_18.PLK2 (NodeNumber=19) [Cable Type=PowerlinkCable, Length=10, Version=1.0.0.3]; PLK2 -> SEG_H_20.PLK1 (NodeNumber=19) [Cable Type=PowerlinkCable, Length=10, Version=1.0.0.3]]
  EnableDNA = on
  EPL_DNA_Head = 0
  EPL_DNA_Predecessor = 20
  DriveConfiguration:
    McTypeID = LLMConfig
  DriveConfiguration/Segment:
    Shape = STRAIGHT105_TO_CIRCULAR
    SegmentReference = SEG_H_19
    StopReaction = UseAssemblySetting
    SpeedFilter = UseAssemblySetting
SEG_H_20 : 8F1I01.AA66.xxxx-1 v1.0.0.2  [PLK1 -> SEG_H_19.PLK2 (NodeNumber=20) [Cable Type=PowerlinkCable, Length=10, Version=1.0.0.3]; PLK2 -> SEG_H_21.PLK1 (NodeNumber=20) [Cable Type=PowerlinkCable, Length=10, Version=1.0.0.3]; PLK3 -> 0AC808.9a.ETH3 (NodeNumber=20) [Cable Type=PowerlinkCable, Length=10, Version=1.0.0.3]]
  EnableDNA = on
  EPL_DNA_Head = 0
  EPL_DNA_HubPort = 0
  EPL_DNA_InPort = 3
  DriveConfiguration:
    McTypeID = LLMConfig
  DriveConfiguration/Segment:
    Shape = STRAIGHT660
    SegmentReference = SEG_H_20
    StopReaction = UseAssemblySetting
    SpeedFilter = UseAssemblySetting
SEG_H_21 : 8F1I01.BA2B.xxxx-1 v1.0.0.2  [PLK1 -> SEG_H_20.PLK2 (NodeNumber=21) [Cable Type=PowerlinkCable, Length=10, Version=1.0.0.3]; PLK2 -> SEG_H_22.PLK1 (NodeNumber=21) [Cable Type=PowerlinkCable, Length=10, Version=1.0.0.3]]
  EnableDNA = on
  EPL_DNA_Head = 0
  EPL_DNA_Predecessor = 20
  EPL_DNA_HubPort = 1
  EPL_DNA_InPort = 2
  DriveConfiguration:
    McTypeID = LLMConfig
  DriveConfiguration/Segment:
    Shape = CIRCULAR_TO_STRAIGHT105
    SegmentReference = SEG_H_21
    StopReaction = UseAssemblySetting
    SpeedFilter = UseAssemblySetting
SEG_H_22 : 8F1I01.BB4B.xxxx-1 v1.0.0.2  [PLK1 -> SEG_H_21.PLK2 (NodeNumber=22) [Cable Type=PowerlinkCable, Length=10, Version=1.0.0.3]; PLK2 -> SEG_H_23.PLK1 (NodeNumber=22) [Cable Type=PowerlinkCable, Length=10, Version=1.0.0.3]]
  EnableDNA = on
  EPL_DNA_Head = 0
  EPL_DNA_Predecessor = 21
  EPL_DNA_HubPort = 1
  EPL_DNA_InPort = 2
  DriveConfiguration:
    McTypeID = LLMConfig
  DriveConfiguration/Segment:
    Shape = CIRCULAR
    SegmentReference = SEG_H_22
    StopReaction = UseAssemblySetting
    SpeedFilter = UseAssemblySetting
SEG_H_23 : 8F1I01.AB2B.xxxx-1 v1.0.0.2  [PLK1 -> SEG_H_22.PLK2 (NodeNumber=23) [Cable Type=PowerlinkCable, Length=10, Version=1.0.0.3]; PLK2 -> SEG_H_24.PLK1 (NodeNumber=23) [Cable Type=PowerlinkCable, Length=10, Version=1.0.0.3]]
  EnableDNA = on
  EPL_DNA_Head = 0
  EPL_DNA_Predecessor = 22
  EPL_DNA_HubPort = 1
  EPL_DNA_InPort = 2
  DriveConfiguration:
    McTypeID = LLMConfig
  DriveConfiguration/Segment:
    Shape = STRAIGHT105_TO_CIRCULAR
    SegmentReference = SEG_H_23
    StopReaction = UseAssemblySetting
    SpeedFilter = UseAssemblySetting
SEG_H_24 : 8F1I01.AA66.xxxx-1 v1.0.0.2  [PLK1 -> SEG_H_23.PLK2 (NodeNumber=24) [Cable Type=PowerlinkCable, Length=10, Version=1.0.0.3]]
  EnableDNA = on
  EPL_DNA_Head = 0
  EPL_DNA_Predecessor = 23
  EPL_DNA_HubPort = 1
  EPL_DNA_InPort = 2
  DriveConfiguration:
    McTypeID = LLMConfig
  DriveConfiguration/Segment:
    Shape = STRAIGHT660
    SegmentReference = SEG_H_24
    StopReaction = UseAssemblySetting
    SpeedFilter = UseAssemblySetting
SEG_I_30 : 8F1I01.AA66.xxxx-1 v1.0.0.2  [PLK2 -> SEG_I_31.PLK1 (NodeNumber=30) [Cable Type=PowerlinkCable, Length=10, Version=1.0.0.3]]
  EnableDNA = on
  EPL_DNA_Head = 0
  EPL_DNA_Predecessor = 31
  EPL_DNA_HubPort = 1
  EPL_DNA_InPort = 2
  DriveConfiguration:
    McTypeID = LLMConfig
  DriveConfiguration/Segment:
    Shape = STRAIGHT660
    SegmentReference = SEG_I_30
    StopReaction = UseAssemblySetting
    SpeedFilter = UseAssemblySetting
SEG_I_31 : 8F1I01.AA66.xxxx-1 v1.0.0.2  [PLK1 -> SEG_I_30.PLK2 (NodeNumber=31) [Cable Type=PowerlinkCable, Length=10, Version=1.0.0.3]; PLK2 -> SEG_I_32.PLK1 (NodeNumber=31) [Cable Type=PowerlinkCable, Length=10, Version=1.0.0.3]]
  EnableDNA = on
  EPL_DNA_Head = 0
  EPL_DNA_Predecessor = 32
  EPL_DNA_HubPort = 1
  EPL_DNA_InPort = 2
  DriveConfiguration:
    McTypeID = LLMConfig
  DriveConfiguration/Segment:
    Shape = STRAIGHT660
    SegmentReference = SEG_I_31
    StopReaction = UseAssemblySetting
    SpeedFilter = UseAssemblySetting
SEG_I_32 : 8F1I01.AA66.xxxx-1 v1.0.0.2  [PLK1 -> SEG_I_31.PLK2 (NodeNumber=32) [Cable Type=PowerlinkCable, Length=10, Version=1.0.0.3]; PLK2 -> SEG_I_33.PLK1 (NodeNumber=32) [Cable Type=PowerlinkCable, Length=10, Version=1.0.0.3]]
  EnableDNA = on
  EPL_DNA_Head = 0
  EPL_DNA_Predecessor = 33
  EPL_DNA_HubPort = 1
  EPL_DNA_InPort = 2
  DriveConfiguration:
    McTypeID = LLMConfig
  DriveConfiguration/Segment:
    Shape = STRAIGHT660
    SegmentReference = SEG_I_32
    StopReaction = UseAssemblySetting
    SpeedFilter = UseAssemblySetting
SEG_I_33 : 8F1I01.AB2B.xxxx-1 v1.0.0.2  [PLK1 -> SEG_I_32.PLK2 (NodeNumber=33) [Cable Type=PowerlinkCable, Length=10, Version=1.0.0.3]; PLK2 -> SEG_I_34.PLK1 (NodeNumber=33) [Cable Type=PowerlinkCable, Length=10, Version=1.0.0.3]]
  EnableDNA = on
  EPL_DNA_Head = 0
  EPL_DNA_Predecessor = 34
  EPL_DNA_HubPort = 1
  EPL_DNA_InPort = 2
  DriveConfiguration:
    McTypeID = LLMConfig
  DriveConfiguration/Segment:
    Shape = STRAIGHT105_TO_CIRCULAR
    SegmentReference = SEG_I_33
    StopReaction = UseAssemblySetting
    SpeedFilter = UseAssemblySetting
SEG_I_34 : 8F1I01.BB4B.xxxx-1 v1.0.0.2  [PLK1 -> SEG_I_33.PLK2 (NodeNumber=34) [Cable Type=PowerlinkCable, Length=10, Version=1.0.0.3]; PLK2 -> SEG_I_35.PLK1 (NodeNumber=34) [Cable Type=PowerlinkCable, Length=10, Version=1.0.0.3]]
  EnableDNA = on
  EPL_DNA_Head = 0
  EPL_DNA_Predecessor = 35
  EPL_DNA_HubPort = 1
  EPL_DNA_InPort = 2
  DriveConfiguration:
    McTypeID = LLMConfig
  DriveConfiguration/Segment:
    Shape = CIRCULAR
    SegmentReference = SEG_I_34
    StopReaction = UseAssemblySetting
    SpeedFilter = UseAssemblySetting
SEG_I_35 : 8F1I01.BA2B.xxxx-1 v1.0.0.2  [PLK1 -> SEG_I_34.PLK2 (NodeNumber=35) [Cable Type=PowerlinkCable, Length=10, Version=1.0.0.3]; PLK3 -> 0AC808.9a.ETH4 (NodeNumber=35) [Cable Type=PowerlinkCable, Length=10, Version=1.0.0.3]]
  EnableDNA = on
  EPL_DNA_Head = 0
  EPL_DNA_HubPort = 0
  EPL_DNA_InPort = 3
  DriveConfiguration:
    McTypeID = LLMConfig
  DriveConfiguration/Segment:
    Shape = CIRCULAR_TO_STRAIGHT105
    SegmentReference = SEG_I_35
    StopReaction = UseAssemblySetting
    SpeedFilter = UseAssemblySetting
SEG_J_36 : 8F1I01.BA2B.xxxx-1 v1.0.0.2  [PLK2 -> SEG_J_37.PLK1 (NodeNumber=55) [Cable Type=PowerlinkCable, Length=10, Version=1.0.0.3]]
  EnableDNA = on
  EPL_DNA_Head = 0
  EPL_DNA_Predecessor = 37
  DriveConfiguration:
    McTypeID = LLMConfig
  DriveConfiguration/Segment:
    Shape = CIRCULAR_TO_STRAIGHT105
    SegmentReference = SEG_J_36
    StopReaction = UseAssemblySetting
    SpeedFilter = UseAssemblySetting
SEG_J_37 : 8F1I01.BB4B.xxxx-1 v1.0.0.2  [PLK1 -> SEG_J_36.PLK2 (NodeNumber=54) [Cable Type=PowerlinkCable, Length=10, Version=1.0.0.3]; PLK2 -> SEG_J_38.PLK1 (NodeNumber=54) [Cable Type=PowerlinkCable, Length=10, Version=1.0.0.3]]
  EnableDNA = on
  EPL_DNA_Head = 0
  EPL_DNA_Predecessor = 38
  DriveConfiguration:
    McTypeID = LLMConfig
  DriveConfiguration/Segment:
    Shape = CIRCULAR
    SegmentReference = SEG_J_37
    StopReaction = UseAssemblySetting
    SpeedFilter = UseAssemblySetting
SEG_J_38 : 8F1I01.AB2B.xxxx-1 v1.0.0.2  [PLK1 -> SEG_J_37.PLK2 (NodeNumber=53) [Cable Type=PowerlinkCable, Length=10, Version=1.0.0.3]; PLK2 -> SEG_J_39.PLK1 (NodeNumber=53) [Cable Type=PowerlinkCable, Length=10, Version=1.0.0.3]]
  EnableDNA = on
  EPL_DNA_Head = 0
  EPL_DNA_Predecessor = 39
  DriveConfiguration:
    McTypeID = LLMConfig
  DriveConfiguration/Segment:
    Shape = STRAIGHT105_TO_CIRCULAR
    SegmentReference = SEG_J_38
    StopReaction = UseAssemblySetting
    SpeedFilter = UseAssemblySetting
SEG_J_39 : 8F1I01.AA66.xxxx-1 v1.0.0.2  [PLK1 -> SEG_J_38.PLK2 (NodeNumber=52) [Cable Type=PowerlinkCable, Length=10, Version=1.0.0.3]; PLK2 -> SEG_J_40.PLK1 (NodeNumber=52) [Cable Type=PowerlinkCable, Length=10, Version=1.0.0.3]; PLK3 -> 0AC808.9c.ETH6 (NodeNumber=52) [Cable Type=PowerlinkCable, Length=10, Version=1.0.0.3]]
  EnableDNA = on
  EPL_DNA_Head = 0
  EPL_DNA_HubPort = 0
  EPL_DNA_InPort = 3
  DriveConfiguration:
    McTypeID = LLMConfig
  DriveConfiguration/Segment:
    Shape = STRAIGHT660
    SegmentReference = SEG_J_39
    StopReaction = UseAssemblySetting
    SpeedFilter = UseAssemblySetting
SEG_J_40 : 8F1I01.BA2B.xxxx-1 v1.0.0.2  [PLK1 -> SEG_J_39.PLK2 (NodeNumber=56) [Cable Type=PowerlinkCable, Length=10, Version=1.0.0.3]; PLK2 -> SEG_J_41.PLK1 (NodeNumber=56) [Cable Type=PowerlinkCable, Length=10, Version=1.0.0.3]]
  EnableDNA = on
  EPL_DNA_Head = 0
  EPL_DNA_Predecessor = 39
  EPL_DNA_HubPort = 1
  EPL_DNA_InPort = 2
  DriveConfiguration:
    McTypeID = LLMConfig
  DriveConfiguration/Segment:
    Shape = CIRCULAR_TO_STRAIGHT105
    SegmentReference = SEG_J_40
    StopReaction = UseAssemblySetting
    SpeedFilter = UseAssemblySetting
SEG_J_41 : 8F1I01.BB4B.xxxx-1 v1.0.0.2  [PLK1 -> SEG_J_40.PLK2 (NodeNumber=57) [Cable Type=PowerlinkCable, Length=10, Version=1.0.0.3]; PLK2 -> SEG_J_42.PLK1 (NodeNumber=57) [Cable Type=PowerlinkCable, Length=10, Version=1.0.0.3]]
  EnableDNA = on
  EPL_DNA_Head = 0
  EPL_DNA_Predecessor = 40
  EPL_DNA_HubPort = 1
  EPL_DNA_InPort = 2
  DriveConfiguration:
    McTypeID = LLMConfig
  DriveConfiguration/Segment:
    Shape = CIRCULAR
    SegmentReference = SEG_J_41
    StopReaction = UseAssemblySetting
    SpeedFilter = UseAssemblySetting
SEG_J_42 : 8F1I01.AB2B.xxxx-1 v1.0.0.2  [PLK1 -> SEG_J_41.PLK2 (NodeNumber=58) [Cable Type=PowerlinkCable, Length=10, Version=1.0.0.3]]
  EnableDNA = on
  EPL_DNA_Head = 0
  EPL_DNA_Predecessor = 41
  EPL_DNA_HubPort = 1
  EPL_DNA_InPort = 2
  DriveConfiguration:
    McTypeID = LLMConfig
  DriveConfiguration/Segment:
    Shape = STRAIGHT105_TO_CIRCULAR
    SegmentReference = SEG_J_42
    StopReaction = UseAssemblySetting
    SpeedFilter = UseAssemblySetting
SEG_K_36 : 8F1I01.BA2B.xxxx-1 v1.0.0.2  [PLK2 -> SEG_K_37.PLK1 (NodeNumber=36) [Cable Type=PowerlinkCable, Length=10, Version=1.0.0.3]]
  EnableDNA = on
  EPL_DNA_Head = 0
  EPL_DNA_Predecessor = 37
  DriveConfiguration:
    McTypeID = LLMConfig
  DriveConfiguration/Segment:
    Shape = CIRCULAR_TO_STRAIGHT105
    SegmentReference = SEG_K_36
    StopReaction = UseAssemblySetting
    SpeedFilter = UseAssemblySetting
SEG_K_37 : 8F1I01.BB4B.xxxx-1 v1.0.0.2  [PLK1 -> SEG_K_36.PLK2 (NodeNumber=37) [Cable Type=PowerlinkCable, Length=10, Version=1.0.0.3]; PLK2 -> SEG_K_38.PLK1 (NodeNumber=37) [Cable Type=PowerlinkCable, Length=10, Version=1.0.0.3]]
  EnableDNA = on
  EPL_DNA_Head = 0
  EPL_DNA_Predecessor = 38
  DriveConfiguration:
    McTypeID = LLMConfig
  DriveConfiguration/Segment:
    Shape = CIRCULAR
    SegmentReference = SEG_K_37
    StopReaction = UseAssemblySetting
    SpeedFilter = UseAssemblySetting
SEG_K_38 : 8F1I01.AB2B.xxxx-1 v1.0.0.2  [PLK1 -> SEG_K_37.PLK2 (NodeNumber=38) [Cable Type=PowerlinkCable, Length=10, Version=1.0.0.3]; PLK2 -> SEG_K_39.PLK1 (NodeNumber=38) [Cable Type=PowerlinkCable, Length=10, Version=1.0.0.3]]
  EnableDNA = on
  EPL_DNA_Head = 0
  EPL_DNA_Predecessor = 39
  DriveConfiguration:
    McTypeID = LLMConfig
  DriveConfiguration/Segment:
    Shape = STRAIGHT105_TO_CIRCULAR
    SegmentReference = SEG_K_38
    StopReaction = UseAssemblySetting
    SpeedFilter = UseAssemblySetting
SEG_K_39 : 8F1I01.AA66.xxxx-1 v1.0.0.2  [PLK1 -> SEG_K_38.PLK2 (NodeNumber=39) [Cable Type=PowerlinkCable, Length=10, Version=1.0.0.3]; PLK2 -> SEG_K_40.PLK1 (NodeNumber=39) [Cable Type=PowerlinkCable, Length=10, Version=1.0.0.3]; PLK3 -> 0AC808.9a.ETH6 (NodeNumber=39) [Cable Type=PowerlinkCable, Length=10, Version=1.0.0.3]]
  EnableDNA = on
  EPL_DNA_Head = 0
  EPL_DNA_HubPort = 0
  EPL_DNA_InPort = 3
  DriveConfiguration:
    McTypeID = LLMConfig
  DriveConfiguration/Segment:
    Shape = STRAIGHT660
    SegmentReference = SEG_K_39
    StopReaction = UseAssemblySetting
    SpeedFilter = UseAssemblySetting
SEG_K_40 : 8F1I01.BA2B.xxxx-1 v1.0.0.2  [PLK1 -> SEG_K_39.PLK2 (NodeNumber=40) [Cable Type=PowerlinkCable, Length=10, Version=1.0.0.3]; PLK2 -> SEG_K_41.PLK1 (NodeNumber=40) [Cable Type=PowerlinkCable, Length=10, Version=1.0.0.3]]
  EnableDNA = on
  EPL_DNA_Head = 0
  EPL_DNA_Predecessor = 39
  EPL_DNA_HubPort = 1
  EPL_DNA_InPort = 2
  DriveConfiguration:
    McTypeID = LLMConfig
  DriveConfiguration/Segment:
    Shape = CIRCULAR_TO_STRAIGHT105
    SegmentReference = SEG_K_40
    StopReaction = UseAssemblySetting
    SpeedFilter = UseAssemblySetting
SEG_K_41 : 8F1I01.BB4B.xxxx-1 v1.0.0.2  [PLK1 -> SEG_K_40.PLK2 (NodeNumber=41) [Cable Type=PowerlinkCable, Length=10, Version=1.0.0.3]; PLK2 -> SEG_K_42.PLK1 (NodeNumber=41) [Cable Type=PowerlinkCable, Length=10, Version=1.0.0.3]]
  EnableDNA = on
  EPL_DNA_Head = 0
  EPL_DNA_Predecessor = 40
  EPL_DNA_HubPort = 1
  EPL_DNA_InPort = 2
  DriveConfiguration:
    McTypeID = LLMConfig
  DriveConfiguration/Segment:
    Shape = CIRCULAR
    SegmentReference = SEG_K_41
    StopReaction = UseAssemblySetting
    SpeedFilter = UseAssemblySetting
SEG_K_42 : 8F1I01.AB2B.xxxx-1 v1.0.0.2  [PLK1 -> SEG_K_41.PLK2 (NodeNumber=42) [Cable Type=PowerlinkCable, Length=10, Version=1.0.0.3]]
  EnableDNA = on
  EPL_DNA_Head = 0
  EPL_DNA_Predecessor = 41
  EPL_DNA_HubPort = 1
  EPL_DNA_InPort = 2
  DriveConfiguration:
    McTypeID = LLMConfig
  DriveConfiguration/Segment:
    Shape = STRAIGHT105_TO_CIRCULAR
    SegmentReference = SEG_K_42
    StopReaction = UseAssemblySetting
    SpeedFilter = UseAssemblySetting
```

### Cfg_PpList.processpointlist - PC/mappMotion/Trak/Cfg_PpList.processpointlist
```
Element ProcessPointList_Outfeed (Type=processpointlist)
  ProcessPoint[0]:
    Name = gMcPrcTrackAOutfeedCam
    SectorRef = gMcSecTrackAOutfeed
    Position = 0.2
    TriggerEventBufferSize = 10
    BarrierFunctionality = On
  ProcessPoint[1]:
    Name = gMcPrcTrackAOutfeedVisTrig
    SectorRef = gMcSecTrackAOutfeed
    Position = 0.793388599952502
    TriggerEventBufferSize = 10
    BarrierFunctionality = Off
  ProcessPoint[2]:
    Name = gMcPrcTrackAOutfeedTangent
    SectorRef = gMcSecTrackAOutfeed
    Position = 0.94900000095367432
    TriggerEventBufferSize = 10
    BarrierFunctionality = Off
  ProcessPoint[3]:
    Name = gMcPrcTrackAOutfeedRelease
    SectorRef = gMcSecTrackAOutfeed
    Position = 1.25
    TriggerEventBufferSize = 10
    BarrierFunctionality = Off
  ProcessPoint[4]:
    Name = gMcPrcTrackAOutfeedBackup1
    SectorRef = gMcSecTrackAOutfeed
    Position = 1.42
    TriggerEventBufferSize = 10
    BarrierFunctionality = Off
  ProcessPoint[5]:
    Name = gMcPrcTrackAOutfeedBackup2
    SectorRef = gMcSecTrackAOutfeed
    Position = 1.52
    TriggerEventBufferSize = 10
    BarrierFunctionality = Off
  ProcessPoint[6]:
    Name = gMcPrcTrackAOutfeedRedirect
    SectorRef = gMcSecTrackAOutfeed
    Position = 0.001
    TriggerEventBufferSize = 10
    BarrierFunctionality = Off
Element ProcessPointList_Infeed (Type=processpointlist)
  ProcessPoint[0]:
    Name = gMcPrcTrackAInfeedCam
    SectorRef = gMcSecTrackAInfeed
    Position = 0.1
    TriggerEventBufferSize = 10
    BarrierFunctionality = On
  ProcessPoint[1]:
    Name = gMcPrcTrackAInfeedVisTrig
    SectorRef = gMcSecTrackAInfeed
    Position = 0.69284954648332477
    TriggerEventBufferSize = 10
    BarrierFunctionality = Off
  ProcessPoint[2]:
    Name = gMcPrcTrackAInfeedTangent
    SectorRef = gMcSecTrackAInfeed
    Position = 0.8609351
    TriggerEventBufferSize = 10
    BarrierFunctionality = Off
  ProcessPoint[3]:
    Name = gMcPrcTrackAInfeedRelease
    SectorRef = gMcSecTrackAInfeed
    Position = 1.05
    TriggerEventBufferSize = 10
    BarrierFunctionality = Off
  ProcessPoint[4]:
    Name = gMcPrcTrackAInfeedBackup1
    SectorRef = gMcSecTrackAInfeed
    Position = 0.1
    PositionRelativeTo = FromEnd
    TriggerEventBufferSize = 10
    BarrierFunctionality = Off
  ProcessPoint[5]:
    Name = gMcPrcTrackAInfeedBackup2
    SectorRef = gMcSecTrackAInfeed
    PositionRelativeTo = FromEnd
    TriggerEventBufferSize = 10
    BarrierFunctionality = Off
  ProcessPoint[6]:
    Name = gMcPrcTrackAInfeedRedirect
    SectorRef = gMcSecTrackAInfeed
    Position = 0.001
    TriggerEventBufferSize = 10
    BarrierFunctionality = Off
Element ProcessPointList_TrackEFlexA (Type=processpointlist)
  ProcessPoint[0]:
    Name = gMcPrcTrackEFlexA0
    SectorRef = gMcSecTrackEFlexA
    Position = 0.001
    TriggerEventBufferSize = 10
    BarrierFunctionality = On
Element ProcessPointList_TrackEFlexB (Type=processpointlist)
  ProcessPoint[0]:
    Name = gMcPrcTrackEFlexB0
    SectorRef = gMcSecTrackEFlexB
    Position = 0.001
    TriggerEventBufferSize = 10
    BarrierFunctionality = On
Element ProcessPointList_TrackEFlexC (Type=processpointlist)
  ProcessPoint[0]:
    Name = gMcPrcTrackEFlexC0
    SectorRef = gMcSecTrackEFlexC
    Position = 0.001
    TriggerEventBufferSize = 10
    BarrierFunctionality = On
Element ProcessPointList_TrackEFlexD (Type=processpointlist)
  ProcessPoint[0]:
    Name = gMcPrcTrackEFlexD0
    SectorRef = gMcSecTrackEFlexD
    Position = 0.001
    TriggerEventBufferSize = 10
    BarrierFunctionality = On
  ProcessPoint[1]:
    Name = gMcPrcTrackFlexLPJ
    SectorRef = gMcSecTrackEFlexD
    Position = 0.120
    TriggerEventBufferSize = 10
    BarrierFunctionality = Off
Element ProcessPointList_TrackEFlexE (Type=processpointlist)
  ProcessPoint[0]:
    Name = gMcPrcTrackEFlexE0
    SectorRef = gMcSecTrackEFlexE
    Position = 0.330
    TriggerEventBufferSize = 10
    BarrierFunctionality = On
  ProcessPoint[1]:
    Name = gMcPrcTrackFlexLPE
    SectorRef = gMcSecTrackEFlexE
    Position = 0.200
    TriggerEventBufferSize = 10
    BarrierFunctionality = Off
Element ProcessPointList_TrackHFlexA (Type=processpointlist)
  ProcessPoint[0]:
    Name = gMcPrcTrackHFlexA0
    SectorRef = gMcSecTrackHFlexA
    Position = 0.001
    TriggerEventBufferSize = 10
    BarrierFunctionality = On
Element ProcessPointList_TrackHFlexB (Type=processpointlist)
  ProcessPoint[0]:
    Name = gMcPrcTrackHFlexB0
    SectorRef = gMcSecTrackHFlexB
    Position = 0.001
    TriggerEventBufferSize = 10
    BarrierFunctionality = On
Element ProcessPointList_TrackHFlexC (Type=processpointlist)
  ProcessPoint[0]:
    Name = gMcPrcTrackHFlexC0
    SectorRef = gMcSecTrackHFlexC
    Position = 0.001
    TriggerEventBufferSize = 10
    BarrierFunctionality = On
Element ProcessPointList_TrackHFlexD (Type=processpointlist)
  ProcessPoint[0]:
    Name = gMcPrcTrackHFlexD0
    SectorRef = gMcSecTrackHFlexD
    Position = 0.001
    TriggerEventBufferSize = 10
    BarrierFunctionality = On
  ProcessPoint[1]:
    Name = gMcPrcTrackFlexLPK
    SectorRef = gMcSecTrackHFlexD
    Position = 0.120
    TriggerEventBufferSize = 10
    BarrierFunctionality = Off
Element ProcessPointList_TrackHFlexE (Type=processpointlist)
  ProcessPoint[0]:
    Name = gMcPrcTrackHFlexE0
    SectorRef = gMcSecTrackHFlexE
    Position = 0.330
    TriggerEventBufferSize = 10
    BarrierFunctionality = On
  ProcessPoint[1]:
    Name = gMcPrcTrackFlexLPH
    SectorRef = gMcSecTrackHFlexE
    Position = 0.200
    TriggerEventBufferSize = 10
    BarrierFunctionality = Off
Element ProcessPointList_OutBuff (Type=processpointlist)
  ProcessPoint[0]:
    Name = gMcPrcTrackAOutBuffStart
    SectorRef = gMcSecTrackAOutBuff
    Position = 0.001
    TriggerEventBufferSize = 10
    BarrierFunctionality = Off
  ProcessPoint[1]:
    Name = gMcPrcTrackAOutBuffEnd
    SectorRef = gMcSecTrackAOutBuff
    Position = 0.001
    PositionRelativeTo = FromEnd
    TriggerEventBufferSize = 10
    BarrierFunctionality = Off
Element ProcessPointList_InBuff (Type=processpointlist)
  ProcessPoint[0]:
    Name = gMcPrcTrackAInBuffStart
    SectorRef = gMcSecTrackAInBuff
    Position = 0.300
    TriggerEventBufferSize = 10
    BarrierFunctionality = Off
  ProcessPoint[1]:
    Name = gMcPrcTrackAInBuffEnd
    SectorRef = gMcSecTrackAInBuff
    Position = 0.001
    PositionRelativeTo = FromEnd
    TriggerEventBufferSize = 10
    BarrierFunctionality = Off
  ProcessPoint[2]:
    Name = gMcPrcTrackAInBarrier
    SectorRef = gMcSecTrackAInBuff
    Position = 0.560
    TriggerEventBufferSize = 10
    BarrierFunctionality = On
Element ProcessPointList_TrackHExMerge (Type=processpointlist)  // PP's for Exclusion zone at trak H between merge A and I
  ProcessPoint[0]:
    Name = gMcPrcH_Merge_A_Start
    SectorRef = gMcSecTrackA_Mer_A
    TriggerEventBufferSize = 10
    BarrierFunctionality = On
  ProcessPoint[1]:
    Name = gMcPrcH_Merge_I_Start
    SectorRef = gMcSecTrackA_Mer_I
    TriggerEventBufferSize = 10
    BarrierFunctionality = On
  ProcessPoint[2]:
    Name = gMcPrcH_Merge_End
    SectorRef = gMcSecTrackA_Mer_A
    PositionRelativeTo = FromEnd
    TriggerEventBufferSize = 10
    BarrierFunctionality = On
Element ProcessPointList_TrackHExDivert (Type=processpointlist)  // PP's for Exclusion zone at trak H between divert at I and K
  ProcessPoint[0]:
    Name = gMcPrcH_Divert_Start
    SectorRef = gMcSecTrackA_Div_I
    TriggerEventBufferSize = 10
    BarrierFunctionality = On
  ProcessPoint[1]:
    Name = gMcPrcH_Divert_I_End
    SectorRef = gMcSecTrackA_Div_I
    PositionRelativeTo = FromEnd
    TriggerEventBufferSize = 10
    BarrierFunctionality = On
  ProcessPoint[2]:
    Name = gMcPrcH_Divert_K_End
    SectorRef = gMcSecTrackA_Div_K
    PositionRelativeTo = FromEnd
    TriggerEventBufferSize = 10
    BarrierFunctionality = On
Element ProcessPointList_TrackEExMerJtoD (Type=processpointlist)  // PP's for Exclusion zone at trak H between merge A and I
  ProcessPoint[0]:
    Name = gMcPrcTrackE_Mer_D_Start
    SectorRef = gMcSecTrackE_Mer_D
    TriggerEventBufferSize = 10
    BarrierFunctionality = On
  ProcessPoint[1]:
    Name = gMcPrcTrackE_Mer_J_Start
    SectorRef = gMcSecTrackE_Mer_J
    TriggerEventBufferSize = 10
    BarrierFunctionality = On
  ProcessPoint[2]:
    Name = gMcPrcTrackE_Mer_D_End
    SectorRef = gMcSecTrackE_Mer_D
    PositionRelativeTo = FromEnd
    TriggerEventBufferSize = 10
    BarrierFunctionality = On
Element ProcessPointList_TrackHExMerKtoG (Type=processpointlist)  // PP's for Exclusion zone at trak H between merge A and I
  ProcessPoint[0]:
    Name = gMcPrcTrackH_Mer_G_Start
    SectorRef = gMcSecTrackH_Mer_G
    TriggerEventBufferSize = 10
    BarrierFunctionality = On
  ProcessPoint[1]:
    Name = gMcPrcTrackH_Mer_K_Start
    SectorRef = gMcSecTrackH_Mer_K
    TriggerEventBufferSize = 10
    BarrierFunctionality = On
  ProcessPoint[2]:
    Name = gMcPrcTrackH_Mer_G_End
    SectorRef = gMcSecTrackH_Mer_G
    PositionRelativeTo = FromEnd
    TriggerEventBufferSize = 10
    BarrierFunctionality = On
Element ProcessPointList_TrackEFlexCnt (Type=processpointlist)
  ProcessPoint[0]:
    Name = gMcSecTrackEFlexCntStart
    SectorRef = gMcSecTrackEFlexCnt
    Position = 0.001
    TriggerEventBufferSize = 10
    BarrierFunctionality = Off
  ProcessPoint[1]:
    Name = gMcSecTrackEFlexCntEnd
    SectorRef = gMcSecTrackEFlexCnt
    Position = 0.001
    PositionRelativeTo = FromEnd
    TriggerEventBufferSize = 10
    BarrierFunctionality = Off
Element ProcessPointList_TrackHFlexCnt (Type=processpointlist)
  ProcessPoint[0]:
    Name = gMcSecTrackHFlexCntStart
    SectorRef = gMcSecTrackHFlexCnt
    Position = 0.001
    TriggerEventBufferSize = 10
    BarrierFunctionality = Off
  ProcessPoint[1]:
    Name = gMcSecTrackHFlexCntEnd
    SectorRef = gMcSecTrackHFlexCnt
    Position = 0.001
    PositionRelativeTo = FromEnd
    TriggerEventBufferSize = 10
    BarrierFunctionality = Off
```

### Cfg_Sec.sector - PC/mappMotion/Trak/Cfg_Sec.sector
```
Element gDivSector_0 (Type=sector)
  Type = Composed
    StartSegment:
      SegmentRef = ::SEG_D_10
      Position = 0.0
    IntermediateSegments
    EndSegment:
      SegmentRef = ::SEG_D_10
      Position = 0.1
Element gDivSector_1 (Type=sector)
  Type = Composed
    StartSegment:
      SegmentRef = ::SEG_E_16
      PositionRelativeTo = FromEnd
      Position = 0.0
    IntermediateSegments
    EndSegment:
      SegmentRef = ::SEG_E_16
      PositionRelativeTo = FromEnd
      Position = 0.1
Element gDivSector_2 (Type=sector)
  Type = Composed
    StartSegment:
      SegmentRef = ::SEG_F_30
      Position = 0.0
    IntermediateSegments
    EndSegment:
      SegmentRef = ::SEG_F_30
      Position = 0.1
Element gDivSector_3 (Type=sector)
  Type = Composed
    StartSegment:
      SegmentRef = ::SEG_F_35
      PositionRelativeTo = FromEnd
      Position = 0.0
    IntermediateSegments
    EndSegment:
      SegmentRef = ::SEG_F_35
      PositionRelativeTo = FromEnd
      Position = 0.1
Element gDivSector_4 (Type=sector)
  Type = Composed
    StartSegment:
      SegmentRef = ::SEG_J_42
      Position = 0.0
    IntermediateSegments
    EndSegment:
      SegmentRef = ::SEG_J_42
      Position = 0.1
Element gDivSector_5 (Type=sector)
  Type = Composed
    StartSegment:
      SegmentRef = ::SEG_H_16
      PositionRelativeTo = FromEnd
      Position = 0.0
    IntermediateSegments
    EndSegment:
      SegmentRef = ::SEG_H_16
      PositionRelativeTo = FromEnd
      Position = 0.1
Element gDivSector_6 (Type=sector)
  Type = Composed
    StartSegment:
      SegmentRef = ::SEG_I_30
      Position = 0.0
    IntermediateSegments
    EndSegment:
      SegmentRef = ::SEG_I_30
      Position = 0.1
Element gDivSector_7 (Type=sector)
  Type = Composed
    StartSegment:
      SegmentRef = ::SEG_I_35
      PositionRelativeTo = FromEnd
      Position = 0.0
    IntermediateSegments
    EndSegment:
      SegmentRef = ::SEG_I_35
      PositionRelativeTo = FromEnd
      Position = 0.1
Element gDivSector_8 (Type=sector)
  Type = Composed
    StartSegment:
      SegmentRef = ::SEG_K_42
      Position = 0.0
    IntermediateSegments
    EndSegment:
      SegmentRef = ::SEG_K_42
      Position = 0.1
```

### Cfg_Sh.shuttlestereotype - PC/mappMotion/Trak/Cfg_Sh.shuttlestereotype
```
Element ShuttleStereotype_1 (Type=shuttlestereotype)
  MeasurementUnit = 5067858
  MeasurementResolution = 0.00001
  MovementLimits = Internal
    VelocityIsReadOnly = 0
    Velocity:
      Velocity = 4.0
    AccelerationIsReadOnly = 0
    Acceleration:
      Acceleration = 20
    DecelerationIsReadOnly = 0
    Deceleration:
      Deceleration = 20
    UpdateMode = Immediately
  JerkFilter = Used
    JerkTime = 0.02
  UserData:
    Size = 4
  CollisionAvoidance:
    InitialModelDimensions = UseExplicitValues
      Length:
        ExtentToFront = 0.029
        ExtentToBack = 0.029
      Width:
        Width = 0.07
```

### Cfg_Trak.assembly - PC/mappMotion/Trak/Cfg_Trak.assembly
```
Element gMcAssembly01 (Type=assembly)
  Tracks:
    TrackSeparation = 0.030
    Track[1]:
      Segments:
        SegmentRef[1] = SEG_A_10
        SegmentRef[2] = SEG_A_11
        SegmentRef[3] = SEG_A_12
        SegmentRef[4] = SEG_A_13
        SegmentRef[5] = SEG_A_14
        SegmentRef[6] = SEG_A_15
        SegmentRef[7] = SEG_A_16
        SegmentRef[8] = SEG_A_17
        SegmentRef[9] = SEG_A_18
        SegmentRef[10] = SEG_A_19
        SegmentRef[11] = SEG_A_20
        SegmentRef[12] = SEG_A_21
        SegmentRef[13] = SEG_A_22
        SegmentRef[14] = SEG_A_23
        SegmentRef[15] = SEG_A_24
        SegmentRef[16] = SEG_A_25
        SegmentRef[17] = SEG_A_26
        SegmentRef[18] = SEG_A_27
        SegmentRef[19] = SEG_A_28
        SegmentRef[20] = SEG_A_29
        SegmentRef[21] = SEG_A_30
        SegmentRef[22] = SEG_A_31
        SegmentRef[23] = SEG_A_32
        SegmentRef[24] = SEG_A_33
        SegmentRef[25] = SEG_A_34
        SegmentRef[26] = SEG_A_35
        SegmentRef[27] = SEG_A_36
        SegmentRef[28] = SEG_A_37
        SegmentRef[29] = SEG_A_38
        SegmentRef[30] = SEG_A_39
      Position = Absolute
        SegmentRef = SEG_A_14
        SegmentCountDirection = RightToLeft
        PositionRelativeTo = FromEnd
        Translation:
          X = 0.0
          Y = 0.0
          Z = 0.0
        Orientation:
          Angle1 = 0.0
          Angle2 = 0.0
          Angle3 = 0.0
    Track[2]:
      Segments:
        SegmentRef[1] = SEG_D_10
        SegmentRef[2] = SEG_D_11
        SegmentRef[3] = SEG_D_12
        SegmentRef[4] = SEG_D_13
        SegmentRef[5] = SEG_D_14
        SegmentRef[6] = SEG_D_15
      Position = RelativeToOne
        TrackSegmentPosition:
          SegmentRef = SEG_D_10
        Base:
          SegmentRef = SEG_A_39
          Position = 0.000621
          PositionRelativeTo = FromEnd
    Track[3]:
      Segments:
        SegmentRef[1] = SEG_E_24
        SegmentRef[2] = SEG_E_23
        SegmentRef[3] = SEG_E_22
        SegmentRef[4] = SEG_E_21
        SegmentRef[5] = SEG_E_20
        SegmentRef[6] = SEG_E_19
        SegmentRef[7] = SEG_E_18
        SegmentRef[8] = SEG_E_17
        SegmentRef[9] = SEG_E_16
      Position = RelativeToOne
        TrackSegmentPosition:
          SegmentRef = SEG_E_16
          PositionRelativeTo = FromEnd
        Base:
          SegmentRef = SEG_D_15
          Position = 0.104015  // 0.1
          PositionRelativeTo = FromEnd
    Track[4]:
      Segments:
        SegmentRef[1] = SEG_F_30
        SegmentRef[2] = SEG_F_31
        SegmentRef[3] = SEG_F_32
        SegmentRef[4] = SEG_F_33
        SegmentRef[5] = SEG_F_34
        SegmentRef[6] = SEG_F_35
        SegmentRef[7] = SEG_G_10
        SegmentRef[8] = SEG_G_11
        SegmentRef[9] = SEG_G_12
        SegmentRef[10] = SEG_G_13
        SegmentRef[11] = SEG_G_14
        SegmentRef[12] = SEG_G_15
      Position = RelativeToTwo
        AlignmentToFirst:
          SegmentRefNewFirst = SEG_F_30
          SegmentRefBaseFirst = ::SEG_E_24
        AlignmentToSecond:
          SegmentRefNewSecond = SEG_F_35
          SegmentRefBaseSecond = SEG_A_35
    Track[5]:
      Segments:
        SegmentRef[1] = SEG_J_42
        SegmentRef[2] = SEG_J_41
        SegmentRef[3] = SEG_J_40
        SegmentRef[4] = SEG_J_39
        SegmentRef[5] = SEG_J_38
        SegmentRef[6] = SEG_J_37
        SegmentRef[7] = SEG_J_36
      Position = RelativeToOne
        TrackSegmentPosition:
          SegmentRef = SEG_J_42
        Base:
          SegmentRef = SEG_D_13
          Position = 0.254651
    Track[6]:
      Segments:
        SegmentRef[1] = SEG_H_24
        SegmentRef[2] = SEG_H_23
        SegmentRef[3] = SEG_H_22
        SegmentRef[4] = SEG_H_21
        SegmentRef[5] = SEG_H_20
        SegmentRef[6] = SEG_H_19
        SegmentRef[7] = SEG_H_18
        SegmentRef[8] = SEG_H_17
        SegmentRef[9] = SEG_H_16
      Position = RelativeToOne
        TrackSegmentPosition:
          SegmentRef = SEG_H_16
          PositionRelativeTo = FromEnd
        Base:
          SegmentRef = SEG_G_15
          Position = 0.106253  // 0.1
          PositionRelativeTo = FromEnd
    Track[7]:
      Segments:
        SegmentRef[1] = SEG_I_30
        SegmentRef[2] = SEG_I_31
        SegmentRef[3] = SEG_I_32
        SegmentRef[4] = SEG_I_33
        SegmentRef[5] = SEG_I_34
        SegmentRef[6] = SEG_I_35
      Position = RelativeToTwo
        AlignmentToFirst:
          SegmentRefNewFirst = SEG_I_30
          SegmentRefBaseFirst = SEG_H_24
        AlignmentToSecond:
          SegmentRefNewSecond = SEG_I_35
          SegmentRefBaseSecond = SEG_A_30
    Track[8]:
      Segments:
        SegmentRef[1] = SEG_K_42
        SegmentRef[2] = SEG_K_41
        SegmentRef[3] = SEG_K_40
        SegmentRef[4] = SEG_K_39
        SegmentRef[5] = SEG_K_38
        SegmentRef[6] = SEG_K_37
        SegmentRef[7] = SEG_K_36
      Position = RelativeToOne
        TrackSegmentPosition:
          SegmentRef = SEG_K_42
          Position = 0
        Base:
          SegmentRef = SEG_G_13
          Position = 0.25575255
  CommonSegmentSettings:
    SegmentSimulationOnPLC = Off
    StopReaction = InductionHalt
    SpeedFilter = Lowpass
      FilterTime = 0.0008
    ControllerParameters:
      DefaultParameter:
        Controller:
          Position:
            ProportionalGain = 200
          Speed:
            ProportionalGain = 150
            IntegrationTime = 0
          FeedForward:
            TotalMass = 1.5
            ForcePositive = 1
            ForceNegative = 1
            SpeedForceFactor = 0
            ForceLoad = 0.0
        MovementErrorLimits:
          PositionError = 0.004
          VelocityError = 50
      AdditionalParameterSets = NotUsed
    ScopeOfErrorReaction = Assembly
    ShuttleIdentificationTime = 0
  Shuttles:
    MaxShuttleCount = 150
    DistanceReserve:
      Collision = 0.002
      ErrorStop = 0.006
    ShuttleStereotypes:
      ShuttleStRef[1] = ShuttleStereotype_1
    MagnetPlateConfigurations:
      ShuttleType[1] = 8F1SA.100.xxxxxx-x
    CollisionAvoidance:
      Strategy = Constant
      MaximumModelDimensions:
        Length:
          ExtentToFront = 0.0355
          ExtentToBack = 0.0355
        Width:
          Width = 0.0705
  Visualization:
    MonitoringPv = ::Vis:ShuttleMon
    ProcessingTaskClass = 8
```

- Safety project (password-protected, skipped)
